LIN {X -0.018,Y -257.062,Z 1664.281,A 0.000,B 0.000,C 90.000,E1 50.598} C_DIS
LIN {X 0.149,Y -245.227,Z 1664.263,A 0.000,B 0.000,C 90.000,E1 47.310} C_DIS
LIN {X -0.032,Y -234.510,Z 1664.245,A 0.000,B 0.000,C 90.000,E1 44.028} C_DIS
LIN {X 0.021,Y -224.506,Z 1664.226,A 0.000,B 0.000,C 90.000,E1 40.620} C_DIS
LIN {X -0.056,Y -216.375,Z 1664.209,A 0.000,B 0.000,C 90.000,E1 37.569} C_DIS
LIN {X 0.091,Y -208.880,Z 1664.191,A 0.000,B 0.000,C 90.000,E1 34.405} C_DIS
LIN {X -0.009,Y -201.954,Z 1664.174,A 0.000,B 0.000,C 90.000,E1 31.258} C_DIS
LIN {X 0.029,Y -195.573,Z 1664.156,A 0.000,B 0.000,C 90.000,E1 28.025} C_DIS
LIN {X -0.014,Y -189.790,Z 1664.138,A 0.000,B 0.000,C 90.000,E1 24.771} C_DIS
LIN {X -0.011,Y -184.718,Z 1664.119,A 0.000,B 0.000,C 90.000,E1 21.461} C_DIS
LIN {X -0.051,Y -180.294,Z 1664.101,A 0.000,B 0.000,C 90.000,E1 18.127} C_DIS
LIN {X 0.041,Y -176.550,Z 1664.082,A 0.000,B 0.000,C 90.000,E1 14.717} C_DIS
LIN {X -0.073,Y -172.830,Z 1664.058,A 0.000,B 0.000,C 90.000,E1 10.489} C_DIS
LIN {X 0.072,Y -169.604,Z 1664.029,A 0.000,B 0.000,C 90.000,E1 5.277} C_DIS
LIN {X -0.060,Y -167.411,Z 1663.993,A 0.000,B 0.000,C 90.000,E1 358.682} C_DIS
LIN {X -0.010,Y -168.408,Z 1663.930,A 0.000,B 0.000,C 90.000,E1 347.353} C_DIS
LIN {X 0.070,Y -171.194,Z 1663.901,A 0.000,B 0.000,C 90.000,E1 342.127} C_DIS
LIN {X -0.005,Y -174.815,Z 1663.877,A 0.000,B 0.000,C 90.000,E1 337.847} C_DIS
LIN {X 0.066,Y -178.691,Z 1663.858,A 0.000,B 0.000,C 90.000,E1 334.409} C_DIS
LIN {X -0.019,Y -183.314,Z 1663.839,A 0.000,B 0.000,C 90.000,E1 331.051} C_DIS
LIN {X -0.041,Y -188.766,Z 1663.821,A 0.000,B 0.000,C 90.000,E1 327.709} C_DIS
LIN {X 0.106,Y -193.563,Z 1663.807,A 0.000,B 0.000,C 90.000,E1 325.182} C_DIS
LIN {X -0.026,Y -198.905,Z 1663.793,A 0.000,B 0.000,C 90.000,E1 322.763} C_DIS
LIN {X 0.074,Y -205.972,Z 1663.777,A 0.000,B 0.000,C 90.000,E1 319.908} C_DIS
LIN {X 0.004,Y -213.943,Z 1663.762,A 0.000,B 0.000,C 90.000,E1 317.148} C_DIS
LIN {X -0.055,Y -222.887,Z 1663.747,A 0.000,B 0.000,C 90.000,E1 314.433} C_DIS
LIN {X 0.034,Y -234.369,Z 1663.730,A 0.000,B 0.000,C 90.000,E1 311.353} C_DIS
LIN {X -0.013,Y -245.664,Z 1663.715,A 0.000,B 0.000,C 90.000,E1 308.749} C_DIS
LIN {X -0.136,Y -256.628,Z 1663.703,A 0.000,B 0.000,C 90.000,E1 306.583} C_DIS
LIN {X -0.013,Y -272.944,Z 1663.687,A 0.000,B 0.000,C 90.000,E1 303.706} C_DIS
LIN {X 0.096,Y -291.059,Z 1663.672,A 0.000,B 0.000,C 90.000,E1 300.924} C_DIS
LIN {X -0.028,Y -310.502,Z 1663.657,A 0.000,B 0.000,C 90.000,E1 298.281} C_DIS
LIN {X -0.059,Y -323.099,Z 1663.648,A 0.000,B 0.000,C 90.000,E1 296.668} C_DIS
LIN {X -0.045,Y -335.406,Z 1663.639,A 0.000,B 0.000,C 90.000,E1 295.079} C_DIS
LIN {X 0.044,Y -350.168,Z 1663.629,A 0.000,B 0.000,C 90.000,E1 293.206} C_DIS
LIN {X -0.102,Y -362.395,Z 1663.621,A 0.000,B 0.000,C 90.000,E1 291.716} C_DIS
LIN {X 0.183,Y -371.921,Z 1663.614,A 0.000,B 0.000,C 90.000,E1 290.482} C_DIS
LIN {X -0.006,Y -378.695,Z 1663.609,A 0.000,B 0.000,C 90.000,E1 289.631} C_DIS
LIN {X -0.131,Y -384.956,Z 1663.604,A 0.000,B 0.000,C 90.000,E1 288.779} C_DIS
LIN {X 0.161,Y -390.546,Z 1663.599,A 0.000,B 0.000,C 90.000,E1 287.873} C_DIS
LIN {X 0.025,Y -395.292,Z 1663.595,A 0.000,B 0.000,C 90.000,E1 287.040} C_DIS
LIN {X -0.133,Y -398.011,Z 1663.592,A 0.000,B 0.000,C 90.000,E1 286.496} C_DIS
LIN {X 0.180,Y -401.321,Z 1663.587,A 0.000,B 0.000,C 90.000,E1 285.607} C_DIS
LIN {X 0.057,Y -403.082,Z 1663.584,A 0.000,B 0.000,C 90.000,E1 285.064} C_DIS
LIN {X -0.167,Y -404.505,Z 1663.581,A 0.000,B 0.000,C 90.000,E1 284.537} C_DIS
LIN {X 0.016,Y -405.481,Z 1663.578,A 0.000,B 0.000,C 90.000,E1 283.953} C_DIS
LIN {X -0.091,Y -406.070,Z 1663.574,A 0.000,B 0.000,C 90.000,E1 283.411} C_DIS
LIN {X 0.108,Y -406.200,Z 1663.571,A 0.000,B 0.000,C 90.000,E1 282.827} C_DIS
LIN {X -0.084,Y -405.886,Z 1663.568,A 0.000,B 0.000,C 90.000,E1 282.299} C_DIS
LIN {X 0.122,Y -405.095,Z 1663.565,A 0.000,B 0.000,C 90.000,E1 281.715} C_DIS
LIN {X -0.071,Y -403.731,Z 1663.562,A 0.000,B 0.000,C 90.000,E1 281.186} C_DIS
LIN {X 0.125,Y -401.822,Z 1663.559,A 0.000,B 0.000,C 90.000,E1 280.602} C_DIS
LIN {X -0.082,Y -399.374,Z 1663.556,A 0.000,B 0.000,C 90.000,E1 280.074} C_DIS
LIN {X 0.018,Y -396.298,Z 1663.553,A 0.000,B 0.000,C 90.000,E1 279.500} C_DIS
LIN {X -0.158,Y -390.804,Z 1663.548,A 0.000,B 0.000,C 90.000,E1 278.681} C_DIS
LIN {X -0.052,Y -384.534,Z 1663.543,A 0.000,B 0.000,C 90.000,E1 277.814} C_DIS
LIN {X -0.008,Y -377.358,Z 1663.539,A 0.000,B 0.000,C 90.000,E1 276.947} C_DIS
LIN {X 0.033,Y -371.956,Z 1663.535,A 0.000,B 0.000,C 90.000,E1 276.372} C_DIS
LIN {X -0.134,Y -366.148,Z 1663.532,A 0.000,B 0.000,C 90.000,E1 275.853} C_DIS
LIN {X -0.023,Y -359.968,Z 1663.530,A 0.000,B 0.000,C 90.000,E1 275.334} C_DIS
LIN {X 0.031,Y -353.523,Z 1663.527,A 0.000,B 0.000,C 90.000,E1 274.878} C_DIS
LIN {X 0.062,Y -347.074,Z 1663.525,A 0.000,B 0.000,C 90.000,E1 274.473} C_DIS
LIN {X -0.043,Y -337.427,Z 1663.522,A 0.000,B 0.000,C 90.000,E1 273.955} C_DIS
LIN {X 0.126,Y -327.816,Z 1663.519,A 0.000,B 0.000,C 90.000,E1 273.440} C_DIS
LIN {X -0.078,Y -318.091,Z 1663.517,A 0.000,B 0.000,C 90.000,E1 273.037} C_DIS
LIN {X -0.021,Y -308.209,Z 1663.515,A 0.000,B 0.000,C 90.000,E1 272.636} C_DIS
LIN {X -0.061,Y -301.352,Z 1663.513,A 0.000,B 0.000,C 90.000,E1 272.407} C_DIS
LIN {X 0.052,Y -294.071,Z 1663.512,A 0.000,B 0.000,C 90.000,E1 272.178} C_DIS
LIN {X 0.045,Y -286.541,Z 1663.511,A 0.000,B 0.000,C 90.000,E1 272.007} C_DIS
LIN {X -0.087,Y -277.923,Z 1663.510,A 0.000,B 0.000,C 90.000,E1 271.892} C_DIS
LIN {X -0.075,Y -267.107,Z 1663.510,A 0.000,B 0.000,C 90.000,E1 271.776} C_DIS
LIN {X -0.077,Y -233.599,Z 1663.509,A 0.000,B 0.000,C 90.000,E1 271.604} C_DIS
LIN {X -0.054,Y -181.975,Z 1663.508,A 0.000,B 0.000,C 90.000,E1 271.375} C_DIS
LIN {X -0.080,Y -181.381,Z 1663.507,A 0.000,B 0.000,C 90.000,E1 271.375} C_DIS
LIN {X -0.030,Y -181.572,Z 1663.502,A 0.000,B 0.000,C 90.000,E1 270.458} C_DIS
LIN {X -0.052,Y -180.906,Z 1663.474,A 0.000,B 0.000,C 90.000,E1 265.412} C_DIS
LIN {X 0.022,Y -180.702,Z 1663.470,A 0.000,B 0.000,C 90.000,E1 264.546} C_DIS
LIN {X -0.076,Y -178.788,Z 1663.442,A 0.000,B 0.000,C 90.000,E1 259.511} C_DIS
LIN {X 0.002,Y -175.834,Z 1663.413,A 0.000,B 0.000,C 90.000,E1 254.393} C_DIS
LIN {X 0.002,Y -172.023,Z 1663.385,A 0.000,B 0.000,C 90.000,E1 249.263} C_DIS
LIN {X -0.022,Y -171.447,Z 1663.380,A 0.000,B 0.000,C 90.000,E1 248.411} C_DIS
LIN {X 0.032,Y -167.682,Z 1663.356,A 0.000,B 0.000,C 90.000,E1 244.076} C_DIS
LIN {X -0.028,Y -166.359,Z 1663.346,A 0.000,B 0.000,C 90.000,E1 242.359} C_DIS
LIN {X -0.035,Y -163.092,Z 1663.327,A 0.000,B 0.000,C 90.000,E1 238.869} C_DIS
LIN {X 0.015,Y -161.036,Z 1663.312,A 0.000,B 0.000,C 90.000,E1 236.215} C_DIS
LIN {X -0.001,Y -157.775,Z 1663.293,A 0.000,B 0.000,C 90.000,E1 232.683} C_DIS
LIN {X 0.063,Y -155.812,Z 1663.278,A 0.000,B 0.000,C 90.000,E1 229.989} C_DIS
LIN {X 0.009,Y -152.063,Z 1663.253,A 0.000,B 0.000,C 90.000,E1 225.526} C_DIS
LIN {X -0.080,Y -150.314,Z 1663.238,A 0.000,B 0.000,C 90.000,E1 222.852} C_DIS
LIN {X 0.058,Y -147.058,Z 1663.213,A 0.000,B 0.000,C 90.000,E1 218.257} C_DIS
LIN {X 0.050,Y -145.634,Z 1663.197,A 0.000,B 0.000,C 90.000,E1 215.518} C_DIS
LIN {X 0.048,Y -143.017,Z 1663.172,A 0.000,B 0.000,C 90.000,E1 210.924} C_DIS
LIN {X -0.022,Y -141.644,Z 1663.151,A 0.000,B 0.000,C 90.000,E1 207.257} C_DIS
LIN {X 0.030,Y -139.440,Z 1663.115,A 0.000,B 0.000,C 90.000,E1 200.737} C_DIS
LIN {X -0.048,Y -139.174,Z 1663.105,A 0.000,B 0.000,C 90.000,E1 198.906} C_DIS
LIN {X -0.020,Y -138.318,Z 1663.053,A 0.000,B 0.000,C 90.000,E1 189.557} C_DIS
LIN {X -0.011,Y -139.471,Z 1663.006,A 0.000,B 0.000,C 90.000,E1 181.146} C_DIS
LIN {X 0.070,Y -141.043,Z 1662.975,A 0.000,B 0.000,C 90.000,E1 175.527} C_DIS
LIN {X 0.024,Y -142.413,Z 1662.960,A 0.000,B 0.000,C 90.000,E1 172.761} C_DIS
LIN {X -0.055,Y -144.647,Z 1662.934,A 0.000,B 0.000,C 90.000,E1 168.173} C_DIS
LIN {X 0.005,Y -147.843,Z 1662.909,A 0.000,B 0.000,C 90.000,E1 163.559} C_DIS
LIN {X -0.052,Y -150.541,Z 1662.888,A 0.000,B 0.000,C 90.000,E1 159.934} C_DIS
LIN {X -0.034,Y -154.007,Z 1662.868,A 0.000,B 0.000,C 90.000,E1 156.305} C_DIS
LIN {X 0.026,Y -157.421,Z 1662.848,A 0.000,B 0.000,C 90.000,E1 152.692} C_DIS
LIN {X 0.049,Y -161.632,Z 1662.829,A 0.000,B 0.000,C 90.000,E1 149.125} C_DIS
LIN {X 0.067,Y -165.828,Z 1662.809,A 0.000,B 0.000,C 90.000,E1 145.595} C_DIS
LIN {X 0.060,Y -170.798,Z 1662.790,A 0.000,B 0.000,C 90.000,E1 142.110} C_DIS
LIN {X -0.023,Y -175.669,Z 1662.771,A 0.000,B 0.000,C 90.000,E1 138.690} C_DIS
LIN {X 0.101,Y -181.282,Z 1662.752,A 0.000,B 0.000,C 90.000,E1 135.243} C_DIS
LIN {X -0.027,Y -186.760,Z 1662.733,A 0.000,B 0.000,C 90.000,E1 131.919} C_DIS
LIN {X 0.045,Y -191.355,Z 1662.719,A 0.000,B 0.000,C 90.000,E1 129.402} C_DIS
LIN {X -0.031,Y -197.192,Z 1662.701,A 0.000,B 0.000,C 90.000,E1 126.137} C_DIS
LIN {X 0.053,Y -200.469,Z 1662.692,A 0.000,B 0.000,C 90.000,E1 124.485} C_DIS
LIN {X 0.025,Y -207.457,Z 1662.671,A 0.000,B 0.000,C 90.000,E1 120.718} C_DIS
LIN {X 0.001,Y -328.831,Z 1662.671,A 0.000,B 0.000,C 90.000,E1 120.718} C_DIS
LIN {X 0.095,Y -335.276,Z 1662.669,A 0.000,B 0.000,C 90.000,E1 120.463} C_DIS
LIN {X 0.140,Y -338.242,Z 1662.668,A 0.000,B 0.000,C 90.000,E1 120.207} C_DIS
LIN {X 0.031,Y -341.943,Z 1662.665,A 0.000,B 0.000,C 90.000,E1 119.745} C_DIS
LIN {X -0.120,Y -343.606,Z 1662.664,A 0.000,B 0.000,C 90.000,E1 119.461} C_DIS
LIN {X -0.117,Y -357.433,Z 1662.647,A 0.000,B 0.000,C 90.000,E1 116.411} C_DIS
LIN {X 0.102,Y -371.411,Z 1662.632,A 0.000,B 0.000,C 90.000,E1 113.695} C_DIS
LIN {X -0.197,Y -385.182,Z 1662.619,A 0.000,B 0.000,C 90.000,E1 111.408} C_DIS
LIN {X 0.071,Y -400.321,Z 1662.606,A 0.000,B 0.000,C 90.000,E1 109.087} C_DIS
LIN {X 0.085,Y -416.932,Z 1662.594,A 0.000,B 0.000,C 90.000,E1 106.858} C_DIS
LIN {X -0.140,Y -435.129,Z 1662.582,A 0.000,B 0.000,C 90.000,E1 104.717} C_DIS
LIN {X 0.160,Y -454.786,Z 1662.570,A 0.000,B 0.000,C 90.000,E1 102.591} C_DIS
LIN {X 0.237,Y -475.081,Z 1662.559,A 0.000,B 0.000,C 90.000,E1 100.658} C_DIS
LIN {X -0.126,Y -501.079,Z 1662.547,A 0.000,B 0.000,C 90.000,E1 98.511} C_DIS
LIN {X 0.196,Y -504.675,Z 1662.545,A 0.000,B 0.000,C 90.000,E1 98.049} C_DIS
LIN {X 0.127,Y -506.032,Z 1662.543,A 0.000,B 0.000,C 90.000,E1 97.814} C_DIS
LIN {X -0.012,Y -507.029,Z 1662.542,A 0.000,B 0.000,C 90.000,E1 97.587} C_DIS
LIN {X -0.192,Y -508.132,Z 1662.539,A 0.000,B 0.000,C 90.000,E1 97.125} C_DIS
LIN {X 0.139,Y -508.201,Z 1662.537,A 0.000,B 0.000,C 90.000,E1 96.606} C_DIS
LIN {X -0.030,Y -507.247,Z 1662.534,A 0.000,B 0.000,C 90.000,E1 96.144} C_DIS
LIN {X -0.197,Y -505.098,Z 1662.531,A 0.000,B 0.000,C 90.000,E1 95.682} C_DIS
LIN {X 0.175,Y -494.734,Z 1662.523,A 0.000,B 0.000,C 90.000,E1 94.188} C_DIS
LIN {X -0.129,Y -484.275,Z 1662.515,A 0.000,B 0.000,C 90.000,E1 92.751} C_DIS
LIN {X -0.148,Y -473.595,Z 1662.507,A 0.000,B 0.000,C 90.000,E1 91.260} C_DIS
LIN {X 0.152,Y -459.135,Z 1662.496,A 0.000,B 0.000,C 90.000,E1 89.198} C_DIS
LIN {X 0.163,Y -448.105,Z 1662.487,A 0.000,B 0.000,C 90.000,E1 87.650} C_DIS
LIN {X -0.016,Y -436.597,Z 1662.478,A 0.000,B 0.000,C 90.000,E1 86.102} C_DIS
LIN {X -0.200,Y -423.089,Z 1662.468,A 0.000,B 0.000,C 90.000,E1 84.261} C_DIS
LIN {X 0.101,Y -404.171,Z 1662.453,A 0.000,B 0.000,C 90.000,E1 81.489} C_DIS
LIN {X -0.040,Y -386.478,Z 1662.437,A 0.000,B 0.000,C 90.000,E1 78.701} C_DIS
LIN {X -0.091,Y -371.265,Z 1662.423,A 0.000,B 0.000,C 90.000,E1 76.117} C_DIS
LIN {X -0.016,Y -356.575,Z 1662.408,A 0.000,B 0.000,C 90.000,E1 73.449} C_DIS
LIN {X -0.003,Y -339.651,Z 1662.390,A 0.000,B 0.000,C 90.000,E1 70.115} C_DIS
LIN {X 0.105,Y -328.061,Z 1662.376,A 0.000,B 0.000,C 90.000,E1 67.614} C_DIS
LIN {X -0.069,Y -315.627,Z 1662.360,A 0.000,B 0.000,C 90.000,E1 64.793} C_DIS
LIN {X -0.198,Y -304.785,Z 1662.345,A 0.000,B 0.000,C 90.000,E1 62.231} C_DIS
LIN {X 0.078,Y -296.635,Z 1662.335,A 0.000,B 0.000,C 90.000,E1 60.205} C_DIS
LIN {X 0.085,Y -288.273,Z 1662.323,A 0.000,B 0.000,C 90.000,E1 58.201} C_DIS
LIN {X 0.086,Y -279.642,Z 1662.312,A 0.000,B 0.000,C 90.000,E1 56.167} C_DIS
LIN {X 0.022,Y -268.032,Z 1662.297,A 0.000,B 0.000,C 90.000,E1 53.417} C_DIS
LIN {X 0.041,Y -255.522,Z 1662.279,A 0.000,B 0.000,C 90.000,E1 50.231} C_DIS
LIN {X -0.023,Y -243.854,Z 1662.261,A 0.000,B 0.000,C 90.000,E1 46.986} C_DIS
LIN {X 0.101,Y -233.249,Z 1662.242,A 0.000,B 0.000,C 90.000,E1 43.623} C_DIS
LIN {X 0.015,Y -224.374,Z 1662.226,A 0.000,B 0.000,C 90.000,E1 40.620} C_DIS
LIN {X 0.108,Y -216.225,Z 1662.209,A 0.000,B 0.000,C 90.000,E1 37.523} C_DIS
LIN {X 0.079,Y -208.720,Z 1662.191,A 0.000,B 0.000,C 90.000,E1 34.405} C_DIS
LIN {X -0.025,Y -201.781,Z 1662.174,A 0.000,B 0.000,C 90.000,E1 31.258} C_DIS
LIN {X 0.011,Y -195.398,Z 1662.156,A 0.000,B 0.000,C 90.000,E1 28.025} C_DIS
LIN {X -0.037,Y -189.641,Z 1662.138,A 0.000,B 0.000,C 90.000,E1 24.771} C_DIS
LIN {X -0.036,Y -184.606,Z 1662.119,A 0.000,B 0.000,C 90.000,E1 21.461} C_DIS
LIN {X -0.021,Y -180.218,Z 1662.101,A 0.000,B 0.000,C 90.000,E1 18.109} C_DIS
LIN {X -0.036,Y -175.705,Z 1662.077,A 0.000,B 0.000,C 90.000,E1 13.883} C_DIS
LIN {X -0.043,Y -172.203,Z 1662.053,A 0.000,B 0.000,C 90.000,E1 9.613} C_DIS
LIN {X 0.034,Y -169.193,Z 1662.025,A 0.000,B 0.000,C 90.000,E1 4.416} C_DIS
LIN {X 0.021,Y -167.142,Z 1661.978,A 0.000,B 0.000,C 90.000,E1 356.045} C_DIS
LIN {X 0.053,Y -168.789,Z 1661.925,A 0.000,B 0.000,C 90.000,E1 346.464} C_DIS
LIN {X 0.074,Y -171.244,Z 1661.901,A 0.000,B 0.000,C 90.000,E1 342.127} C_DIS
LIN {X 0.000,Y -174.891,Z 1661.877,A 0.000,B 0.000,C 90.000,E1 337.847} C_DIS
LIN {X 0.073,Y -178.787,Z 1661.858,A 0.000,B 0.000,C 90.000,E1 334.409} C_DIS
LIN {X -0.009,Y -183.433,Z 1661.839,A 0.000,B 0.000,C 90.000,E1 331.051} C_DIS
LIN {X -0.027,Y -188.918,Z 1661.821,A 0.000,B 0.000,C 90.000,E1 327.709} C_DIS
LIN {X -0.036,Y -193.733,Z 1661.807,A 0.000,B 0.000,C 90.000,E1 325.229} C_DIS
LIN {X -0.006,Y -199.082,Z 1661.793,A 0.000,B 0.000,C 90.000,E1 322.763} C_DIS
LIN {X 0.100,Y -206.138,Z 1661.777,A 0.000,B 0.000,C 90.000,E1 319.908} C_DIS
LIN {X 0.033,Y -214.113,Z 1661.762,A 0.000,B 0.000,C 90.000,E1 317.148} C_DIS
LIN {X -0.021,Y -223.045,Z 1661.747,A 0.000,B 0.000,C 90.000,E1 314.433} C_DIS
LIN {X -0.080,Y -234.501,Z 1661.730,A 0.000,B 0.000,C 90.000,E1 311.391} C_DIS
LIN {X 0.032,Y -245.793,Z 1661.715,A 0.000,B 0.000,C 90.000,E1 308.749} C_DIS
LIN {X -0.103,Y -254.812,Z 1661.705,A 0.000,B 0.000,C 90.000,E1 306.950} C_DIS
LIN {X 0.064,Y -268.784,Z 1661.691,A 0.000,B 0.000,C 90.000,E1 304.405} C_DIS
LIN {X -0.125,Y -284.119,Z 1661.678,A 0.000,B 0.000,C 90.000,E1 302.005} C_DIS
LIN {X -0.034,Y -300.650,Z 1661.665,A 0.000,B 0.000,C 90.000,E1 299.617} C_DIS
LIN {X 0.029,Y -318.190,Z 1661.652,A 0.000,B 0.000,C 90.000,E1 297.308} C_DIS
LIN {X -0.073,Y -333.022,Z 1661.641,A 0.000,B 0.000,C 90.000,E1 295.412} C_DIS
LIN {X 0.113,Y -347.706,Z 1661.631,A 0.000,B 0.000,C 90.000,E1 293.515} C_DIS
LIN {X -0.078,Y -359.926,Z 1661.622,A 0.000,B 0.000,C 90.000,E1 292.025} C_DIS
LIN {X -0.083,Y -371.883,Z 1661.614,A 0.000,B 0.000,C 90.000,E1 290.536} C_DIS
LIN {X 0.076,Y -378.655,Z 1661.609,A 0.000,B 0.000,C 90.000,E1 289.631} C_DIS
LIN {X -0.047,Y -384.908,Z 1661.604,A 0.000,B 0.000,C 90.000,E1 288.779} C_DIS
LIN {X -0.126,Y -390.518,Z 1661.599,A 0.000,B 0.000,C 90.000,E1 287.928} C_DIS
LIN {X 0.110,Y -395.292,Z 1661.595,A 0.000,B 0.000,C 90.000,E1 287.040} C_DIS
LIN {X -0.047,Y -398.020,Z 1661.592,A 0.000,B 0.000,C 90.000,E1 286.496} C_DIS
LIN {X -0.120,Y -401.353,Z 1661.587,A 0.000,B 0.000,C 90.000,E1 285.662} C_DIS
LIN {X 0.144,Y -403.152,Z 1661.584,A 0.000,B 0.000,C 90.000,E1 285.064} C_DIS
LIN {X -0.079,Y -404.572,Z 1661.581,A 0.000,B 0.000,C 90.000,E1 284.537} C_DIS
LIN {X 0.104,Y -405.619,Z 1661.578,A 0.000,B 0.000,C 90.000,E1 283.953} C_DIS
LIN {X -0.002,Y -406.199,Z 1661.574,A 0.000,B 0.000,C 90.000,E1 283.411} C_DIS
LIN {X 0.198,Y -406.365,Z 1661.571,A 0.000,B 0.000,C 90.000,E1 282.827} C_DIS
LIN {X 0.007,Y -406.061,Z 1661.568,A 0.000,B 0.000,C 90.000,E1 282.299} C_DIS
LIN {X -0.184,Y -405.249,Z 1661.565,A 0.000,B 0.000,C 90.000,E1 281.771} C_DIS
LIN {X 0.020,Y -403.898,Z 1661.562,A 0.000,B 0.000,C 90.000,E1 281.186} C_DIS
LIN {X -0.177,Y -402.005,Z 1661.559,A 0.000,B 0.000,C 90.000,E1 280.658} C_DIS
LIN {X 0.011,Y -399.538,Z 1661.556,A 0.000,B 0.000,C 90.000,E1 280.074} C_DIS
LIN {X 0.111,Y -396.458,Z 1661.553,A 0.000,B 0.000,C 90.000,E1 279.500} C_DIS
LIN {X -0.065,Y -390.923,Z 1661.548,A 0.000,B 0.000,C 90.000,E1 278.681} C_DIS
LIN {X 0.042,Y -384.616,Z 1661.543,A 0.000,B 0.000,C 90.000,E1 277.814} C_DIS
LIN {X 0.084,Y -377.417,Z 1661.539,A 0.000,B 0.000,C 90.000,E1 276.947} C_DIS
LIN {X 0.119,Y -371.993,Z 1661.536,A 0.000,B 0.000,C 90.000,E1 276.372} C_DIS
LIN {X -0.064,Y -366.160,Z 1661.532,A 0.000,B 0.000,C 90.000,E1 275.853} C_DIS
LIN {X 0.051,Y -359.946,Z 1661.530,A 0.000,B 0.000,C 90.000,E1 275.334} C_DIS
LIN {X 0.125,Y -353.500,Z 1661.527,A 0.000,B 0.000,C 90.000,E1 274.878} C_DIS
LIN {X 0.080,Y -343.781,Z 1661.524,A 0.000,B 0.000,C 90.000,E1 274.302} C_DIS
LIN {X -0.132,Y -334.628,Z 1661.521,A 0.000,B 0.000,C 90.000,E1 273.841} C_DIS
LIN {X 0.079,Y -324.911,Z 1661.519,A 0.000,B 0.000,C 90.000,E1 273.326} C_DIS
LIN {X -0.052,Y -315.071,Z 1661.516,A 0.000,B 0.000,C 90.000,E1 272.922} C_DIS
LIN {X 0.061,Y -304.968,Z 1661.514,A 0.000,B 0.000,C 90.000,E1 272.522} C_DIS
LIN {X 0.103,Y -297.928,Z 1661.513,A 0.000,B 0.000,C 90.000,E1 272.293} C_DIS
LIN {X -0.025,Y -290.295,Z 1661.512,A 0.000,B 0.000,C 90.000,E1 272.121} C_DIS
LIN {X 0.019,Y -281.682,Z 1661.511,A 0.000,B 0.000,C 90.000,E1 271.949} C_DIS
LIN {X -0.034,Y -272.063,Z 1661.510,A 0.000,B 0.000,C 90.000,E1 271.835} C_DIS
LIN {X -0.069,Y -243.458,Z 1661.509,A 0.000,B 0.000,C 90.000,E1 271.661} C_DIS
LIN {X 0.071,Y -190.113,Z 1661.508,A 0.000,B 0.000,C 90.000,E1 271.375} C_DIS
LIN {X 0.009,Y -183.846,Z 1661.508,A 0.000,B 0.000,C 90.000,E1 271.375} C_DIS
LIN {X -0.011,Y -181.377,Z 1661.508,A 0.000,B 0.000,C 90.000,E1 271.375} C_DIS
LIN {X 0.042,Y -181.579,Z 1661.502,A 0.000,B 0.000,C 90.000,E1 270.344} C_DIS
LIN {X 0.046,Y -180.887,Z 1661.473,A 0.000,B 0.000,C 90.000,E1 265.122} C_DIS
LIN {X -0.070,Y -179.009,Z 1661.445,A 0.000,B 0.000,C 90.000,E1 260.095} C_DIS
LIN {X 0.024,Y -178.625,Z 1661.440,A 0.000,B 0.000,C 90.000,E1 259.218} C_DIS
LIN {X -0.078,Y -175.677,Z 1661.412,A 0.000,B 0.000,C 90.000,E1 254.157} C_DIS
LIN {X -0.065,Y -172.393,Z 1661.388,A 0.000,B 0.000,C 90.000,E1 249.880} C_DIS
LIN {X -0.049,Y -171.199,Z 1661.379,A 0.000,B 0.000,C 90.000,E1 248.156} C_DIS
LIN {X 0.002,Y -167.487,Z 1661.355,A 0.000,B 0.000,C 90.000,E1 243.819} C_DIS
LIN {X 0.010,Y -166.883,Z 1661.350,A 0.000,B 0.000,C 90.000,E1 242.948} C_DIS
LIN {X 0.001,Y -162.190,Z 1661.321,A 0.000,B 0.000,C 90.000,E1 237.709} C_DIS
LIN {X -0.032,Y -160.758,Z 1661.311,A 0.000,B 0.000,C 90.000,E1 235.960} C_DIS
LIN {X 0.036,Y -157.556,Z 1661.291,A 0.000,B 0.000,C 90.000,E1 232.396} C_DIS
LIN {X -0.025,Y -155.585,Z 1661.276,A 0.000,B 0.000,C 90.000,E1 229.747} C_DIS
LIN {X 0.027,Y -151.869,Z 1661.251,A 0.000,B 0.000,C 90.000,E1 225.243} C_DIS
LIN {X 0.040,Y -150.093,Z 1661.236,A 0.000,B 0.000,C 90.000,E1 222.528} C_DIS
LIN {X -0.043,Y -146.893,Z 1661.211,A 0.000,B 0.000,C 90.000,E1 218.016} C_DIS
LIN {X 0.062,Y -145.480,Z 1661.196,A 0.000,B 0.000,C 90.000,E1 215.231} C_DIS
LIN {X -0.022,Y -142.890,Z 1661.170,A 0.000,B 0.000,C 90.000,E1 210.669} C_DIS
LIN {X 0.035,Y -141.509,Z 1661.150,A 0.000,B 0.000,C 90.000,E1 206.950} C_DIS
LIN {X -0.047,Y -139.391,Z 1661.114,A 0.000,B 0.000,C 90.000,E1 200.482} C_DIS
LIN {X 0.004,Y -139.099,Z 1661.103,A 0.000,B 0.000,C 90.000,E1 198.598} C_DIS
LIN {X -0.005,Y -138.354,Z 1661.057,A 0.000,B 0.000,C 90.000,E1 190.197} C_DIS
LIN {X -0.011,Y -139.515,Z 1661.005,A 0.000,B 0.000,C 90.000,E1 180.859} C_DIS
LIN {X -0.071,Y -141.165,Z 1660.974,A 0.000,B 0.000,C 90.000,E1 175.298} C_DIS
LIN {X 0.041,Y -142.545,Z 1660.958,A 0.000,B 0.000,C 90.000,E1 172.470} C_DIS
LIN {X -0.034,Y -144.818,Z 1660.933,A 0.000,B 0.000,C 90.000,E1 167.881} C_DIS
LIN {X -0.047,Y -147.440,Z 1660.912,A 0.000,B 0.000,C 90.000,E1 164.212} C_DIS
LIN {X -0.018,Y -150.020,Z 1660.892,A 0.000,B 0.000,C 90.000,E1 160.550} C_DIS
LIN {X -0.012,Y -153.355,Z 1660.872,A 0.000,B 0.000,C 90.000,E1 156.922} C_DIS
LIN {X 0.037,Y -155.888,Z 1660.857,A 0.000,B 0.000,C 90.000,E1 154.204} C_DIS
LIN {X -0.064,Y -159.747,Z 1660.837,A 0.000,B 0.000,C 90.000,E1 150.667} C_DIS
LIN {X 0.002,Y -161.986,Z 1660.827,A 0.000,B 0.000,C 90.000,E1 148.869} C_DIS
LIN {X 0.021,Y -166.178,Z 1660.807,A 0.000,B 0.000,C 90.000,E1 145.341} C_DIS
LIN {X 0.014,Y -171.193,Z 1660.788,A 0.000,B 0.000,C 90.000,E1 141.859} C_DIS
LIN {X 0.044,Y -176.075,Z 1660.769,A 0.000,B 0.000,C 90.000,E1 138.405} C_DIS
LIN {X -0.093,Y -180.334,Z 1660.755,A 0.000,B 0.000,C 90.000,E1 135.891} C_DIS
LIN {X 0.015,Y -185.744,Z 1660.736,A 0.000,B 0.000,C 90.000,E1 132.486} C_DIS
LIN {X -0.071,Y -190.355,Z 1660.722,A 0.000,B 0.000,C 90.000,E1 130.011} C_DIS
LIN {X -0.025,Y -197.680,Z 1660.699,A 0.000,B 0.000,C 90.000,E1 125.884} C_DIS
LIN {X 0.017,Y -200.932,Z 1660.690,A 0.000,B 0.000,C 90.000,E1 124.246} C_DIS
LIN {X -0.009,Y -207.317,Z 1660.671,A 0.000,B 0.000,C 90.000,E1 120.797} C_DIS
LIN {X 0.051,Y -207.383,Z 1660.671,A 0.000,B 0.000,C 90.000,E1 120.747} C_DIS
LIN {X 0.036,Y -328.953,Z 1660.671,A 0.000,B 0.000,C 90.000,E1 120.747} C_DIS
LIN {X 0.114,Y -329.958,Z 1660.671,A 0.000,B 0.000,C 90.000,E1 120.718} C_DIS
LIN {X 0.136,Y -335.536,Z 1660.669,A 0.000,B 0.000,C 90.000,E1 120.463} C_DIS
LIN {X -0.134,Y -338.393,Z 1660.668,A 0.000,B 0.000,C 90.000,E1 120.256} C_DIS
LIN {X -0.073,Y -342.089,Z 1660.665,A 0.000,B 0.000,C 90.000,E1 119.745} C_DIS
LIN {X 0.074,Y -343.680,Z 1660.663,A 0.000,B 0.000,C 90.000,E1 119.411} C_DIS
LIN {X 0.057,Y -356.036,Z 1660.648,A 0.000,B 0.000,C 90.000,E1 116.668} C_DIS
LIN {X -0.090,Y -369.848,Z 1660.633,A 0.000,B 0.000,C 90.000,E1 114.003} C_DIS
LIN {X -0.080,Y -383.463,Z 1660.620,A 0.000,B 0.000,C 90.000,E1 111.663} C_DIS
LIN {X -0.221,Y -398.435,Z 1660.608,A 0.000,B 0.000,C 90.000,E1 109.396} C_DIS
LIN {X -0.138,Y -414.866,Z 1660.595,A 0.000,B 0.000,C 90.000,E1 107.149} C_DIS
LIN {X -0.012,Y -432.869,Z 1660.583,A 0.000,B 0.000,C 90.000,E1 104.954} C_DIS
LIN {X 0.180,Y -452.393,Z 1660.571,A 0.000,B 0.000,C 90.000,E1 102.827} C_DIS
LIN {X 0.099,Y -472.623,Z 1660.561,A 0.000,B 0.000,C 90.000,E1 100.894} C_DIS
LIN {X -0.103,Y -496.009,Z 1660.549,A 0.000,B 0.000,C 90.000,E1 98.916} C_DIS
LIN {X -0.235,Y -501.157,Z 1660.547,A 0.000,B 0.000,C 90.000,E1 98.511} C_DIS
LIN {X 0.042,Y -504.671,Z 1660.545,A 0.000,B 0.000,C 90.000,E1 98.049} C_DIS
LIN {X -0.027,Y -505.980,Z 1660.543,A 0.000,B 0.000,C 90.000,E1 97.814} C_DIS
LIN {X -0.166,Y -506.937,Z 1660.542,A 0.000,B 0.000,C 90.000,E1 97.587} C_DIS
LIN {X 0.158,Y -507.974,Z 1660.539,A 0.000,B 0.000,C 90.000,E1 97.068} C_DIS
LIN {X -0.016,Y -507.982,Z 1660.537,A 0.000,B 0.000,C 90.000,E1 96.606} C_DIS
LIN {X -0.185,Y -506.962,Z 1660.534,A 0.000,B 0.000,C 90.000,E1 96.144} C_DIS
LIN {X 0.260,Y -506.020,Z 1660.533,A 0.000,B 0.000,C 90.000,E1 95.853} C_DIS
LIN {X 0.149,Y -504.729,Z 1660.531,A 0.000,B 0.000,C 90.000,E1 95.625} C_DIS
LIN {X -0.090,Y -492.600,Z 1660.522,A 0.000,B 0.000,C 90.000,E1 93.955} C_DIS
LIN {X 0.029,Y -482.137,Z 1660.514,A 0.000,B 0.000,C 90.000,E1 92.465} C_DIS
LIN {X -0.029,Y -471.413,Z 1660.505,A 0.000,B 0.000,C 90.000,E1 90.974} C_DIS
LIN {X -0.021,Y -458.773,Z 1660.495,A 0.000,B 0.000,C 90.000,E1 89.198} C_DIS
LIN {X -0.012,Y -447.719,Z 1660.487,A 0.000,B 0.000,C 90.000,E1 87.650} C_DIS
LIN {X -0.193,Y -436.172,Z 1660.478,A 0.000,B 0.000,C 90.000,E1 86.102} C_DIS
LIN {X -0.076,Y -424.584,Z 1660.469,A 0.000,B 0.000,C 90.000,E1 84.489} C_DIS
LIN {X -0.189,Y -405.561,Z 1660.454,A 0.000,B 0.000,C 90.000,E1 81.781} C_DIS
LIN {X 0.175,Y -387.752,Z 1660.439,A 0.000,B 0.000,C 90.000,E1 78.926} C_DIS
LIN {X 0.065,Y -374.151,Z 1660.426,A 0.000,B 0.000,C 90.000,E1 76.645} C_DIS
LIN {X -0.189,Y -360.966,Z 1660.413,A 0.000,B 0.000,C 90.000,E1 74.338} C_DIS
LIN {X 0.172,Y -345.237,Z 1660.396,A 0.000,B 0.000,C 90.000,E1 71.275} C_DIS
LIN {X -0.034,Y -331.952,Z 1660.381,A 0.000,B 0.000,C 90.000,E1 68.539} C_DIS
LIN {X 0.137,Y -317.926,Z 1660.363,A 0.000,B 0.000,C 90.000,E1 65.357} C_DIS
LIN {X 0.017,Y -308.426,Z 1660.351,A 0.000,B 0.000,C 90.000,E1 63.127} C_DIS
LIN {X -0.024,Y -298.982,Z 1660.338,A 0.000,B 0.000,C 90.000,E1 60.845} C_DIS
LIN {X -0.115,Y -290.680,Z 1660.327,A 0.000,B 0.000,C 90.000,E1 58.869} C_DIS
LIN {X -0.060,Y -282.122,Z 1660.316,A 0.000,B 0.000,C 90.000,E1 56.834} C_DIS
LIN {X 0.081,Y -271.922,Z 1660.302,A 0.000,B 0.000,C 90.000,E1 54.402} C_DIS
LIN {X -0.007,Y -260.592,Z 1660.287,A 0.000,B 0.000,C 90.000,E1 51.618} C_DIS
LIN {X -0.070,Y -248.599,Z 1660.269,A 0.000,B 0.000,C 90.000,E1 48.405} C_DIS
LIN {X 0.020,Y -237.594,Z 1660.250,A 0.000,B 0.000,C 90.000,E1 45.081} C_DIS
LIN {X 0.031,Y -228.427,Z 1660.234,A 0.000,B 0.000,C 90.000,E1 42.081} C_DIS
LIN {X 0.013,Y -219.921,Z 1660.217,A 0.000,B 0.000,C 90.000,E1 39.036} C_DIS
LIN {X 0.028,Y -212.085,Z 1660.200,A 0.000,B 0.000,C 90.000,E1 35.931} C_DIS
LIN {X 0.119,Y -204.857,Z 1660.182,A 0.000,B 0.000,C 90.000,E1 32.752} C_DIS
LIN {X -0.016,Y -198.220,Z 1660.164,A 0.000,B 0.000,C 90.000,E1 29.589} C_DIS
LIN {X -0.081,Y -192.191,Z 1660.146,A 0.000,B 0.000,C 90.000,E1 26.360} C_DIS
LIN {X 0.061,Y -186.832,Z 1660.128,A 0.000,B 0.000,C 90.000,E1 23.025} C_DIS
LIN {X 0.029,Y -182.155,Z 1660.109,A 0.000,B 0.000,C 90.000,E1 19.704} C_DIS
LIN {X 0.099,Y -178.184,Z 1660.091,A 0.000,B 0.000,C 90.000,E1 16.315} C_DIS
LIN {X -0.065,Y -174.163,Z 1660.067,A 0.000,B 0.000,C 90.000,E1 12.119} C_DIS
LIN {X -0.013,Y -171.065,Z 1660.043,A 0.000,B 0.000,C 90.000,E1 7.814} C_DIS
LIN {X -0.031,Y -168.499,Z 1660.015,A 0.000,B 0.000,C 90.000,E1 2.636} C_DIS
LIN {X -0.017,Y -167.124,Z 1659.968,A 0.000,B 0.000,C 90.000,E1 354.318} C_DIS
LIN {X 0.056,Y -168.825,Z 1659.925,A 0.000,B 0.000,C 90.000,E1 346.464} C_DIS
LIN {X 0.043,Y -171.926,Z 1659.896,A 0.000,B 0.000,C 90.000,E1 341.275} C_DIS
LIN {X 0.057,Y -175.869,Z 1659.872,A 0.000,B 0.000,C 90.000,E1 336.975} C_DIS
LIN {X -0.009,Y -179.979,Z 1659.853,A 0.000,B 0.000,C 90.000,E1 333.589} C_DIS
LIN {X 0.019,Y -184.867,Z 1659.834,A 0.000,B 0.000,C 90.000,E1 330.205} C_DIS
LIN {X -0.024,Y -190.585,Z 1659.816,A 0.000,B 0.000,C 90.000,E1 326.882} C_DIS
LIN {X 0.021,Y -197.407,Z 1659.798,A 0.000,B 0.000,C 90.000,E1 323.577} C_DIS
LIN {X 0.080,Y -204.208,Z 1659.782,A 0.000,B 0.000,C 90.000,E1 320.723} C_DIS
LIN {X -0.013,Y -211.919,Z 1659.766,A 0.000,B 0.000,C 90.000,E1 317.957} C_DIS
LIN {X -0.123,Y -220.528,Z 1659.751,A 0.000,B 0.000,C 90.000,E1 315.243} C_DIS
LIN {X 0.061,Y -231.680,Z 1659.734,A 0.000,B 0.000,C 90.000,E1 312.123} C_DIS
LIN {X -0.022,Y -240.921,Z 1659.722,A 0.000,B 0.000,C 90.000,E1 309.886} C_DIS
LIN {X 0.077,Y -251.190,Z 1659.709,A 0.000,B 0.000,C 90.000,E1 307.649} C_DIS
LIN {X -0.053,Y -264.715,Z 1659.695,A 0.000,B 0.000,C 90.000,E1 305.152} C_DIS
LIN {X -0.019,Y -281.884,Z 1659.680,A 0.000,B 0.000,C 90.000,E1 302.339} C_DIS
LIN {X 0.033,Y -298.288,Z 1659.666,A 0.000,B 0.000,C 90.000,E1 299.951} C_DIS
LIN {X -0.048,Y -318.256,Z 1659.652,A 0.000,B 0.000,C 90.000,E1 297.334} C_DIS
LIN {X 0.040,Y -330.588,Z 1659.643,A 0.000,B 0.000,C 90.000,E1 295.720} C_DIS
LIN {X 0.048,Y -342.808,Z 1659.634,A 0.000,B 0.000,C 90.000,E1 294.155} C_DIS
LIN {X -0.077,Y -355.066,Z 1659.626,A 0.000,B 0.000,C 90.000,E1 292.642} C_DIS
LIN {X 0.186,Y -367.110,Z 1659.617,A 0.000,B 0.000,C 90.000,E1 291.099} C_DIS
LIN {X -0.045,Y -374.152,Z 1659.612,A 0.000,B 0.000,C 90.000,E1 290.248} C_DIS
LIN {X -0.209,Y -380.732,Z 1659.608,A 0.000,B 0.000,C 90.000,E1 289.396} C_DIS
LIN {X 0.043,Y -386.803,Z 1659.603,A 0.000,B 0.000,C 90.000,E1 288.489} C_DIS
LIN {X -0.007,Y -392.170,Z 1659.598,A 0.000,B 0.000,C 90.000,E1 287.638} C_DIS
LIN {X -0.134,Y -396.718,Z 1659.593,A 0.000,B 0.000,C 90.000,E1 286.804} C_DIS
LIN {X 0.100,Y -399.271,Z 1659.590,A 0.000,B 0.000,C 90.000,E1 286.205} C_DIS
LIN {X -0.033,Y -401.445,Z 1659.587,A 0.000,B 0.000,C 90.000,E1 285.662} C_DIS
LIN {X 0.127,Y -403.230,Z 1659.584,A 0.000,B 0.000,C 90.000,E1 285.079} C_DIS
LIN {X 0.010,Y -404.661,Z 1659.581,A 0.000,B 0.000,C 90.000,E1 284.537} C_DIS
LIN {X -0.201,Y -405.731,Z 1659.578,A 0.000,B 0.000,C 90.000,E1 284.008} C_DIS
LIN {X 0.088,Y -406.321,Z 1659.575,A 0.000,B 0.000,C 90.000,E1 283.411} C_DIS
LIN {X -0.107,Y -406.514,Z 1659.572,A 0.000,B 0.000,C 90.000,E1 282.883} C_DIS
LIN {X 0.098,Y -406.216,Z 1659.568,A 0.000,B 0.000,C 90.000,E1 282.299} C_DIS
LIN {X -0.092,Y -405.417,Z 1659.565,A 0.000,B 0.000,C 90.000,E1 281.771} C_DIS
LIN {X 0.113,Y -404.101,Z 1659.562,A 0.000,B 0.000,C 90.000,E1 281.186} C_DIS
LIN {X -0.084,Y -402.232,Z 1659.559,A 0.000,B 0.000,C 90.000,E1 280.658} C_DIS
LIN {X 0.105,Y -399.741,Z 1659.556,A 0.000,B 0.000,C 90.000,E1 280.074} C_DIS
LIN {X -0.186,Y -396.645,Z 1659.553,A 0.000,B 0.000,C 90.000,E1 279.557} C_DIS
LIN {X 0.030,Y -391.017,Z 1659.548,A 0.000,B 0.000,C 90.000,E1 278.681} C_DIS
LIN {X 0.136,Y -384.673,Z 1659.544,A 0.000,B 0.000,C 90.000,E1 277.814} C_DIS
LIN {X 0.177,Y -377.484,Z 1659.539,A 0.000,B 0.000,C 90.000,E1 276.947} C_DIS
LIN {X -0.132,Y -372.098,Z 1659.536,A 0.000,B 0.000,C 90.000,E1 276.429} C_DIS
LIN {X 0.122,Y -366.377,Z 1659.533,A 0.000,B 0.000,C 90.000,E1 275.853} C_DIS
LIN {X -0.083,Y -360.220,Z 1659.530,A 0.000,B 0.000,C 90.000,E1 275.391} C_DIS
LIN {X -0.008,Y -353.811,Z 1659.527,A 0.000,B 0.000,C 90.000,E1 274.935} C_DIS
LIN {X -0.063,Y -344.090,Z 1659.524,A 0.000,B 0.000,C 90.000,E1 274.359} C_DIS
LIN {X -0.046,Y -334.607,Z 1659.521,A 0.000,B 0.000,C 90.000,E1 273.841} C_DIS
LIN {X 0.154,Y -324.864,Z 1659.519,A 0.000,B 0.000,C 90.000,E1 273.326} C_DIS
LIN {X 0.004,Y -314.933,Z 1659.516,A 0.000,B 0.000,C 90.000,E1 272.922} C_DIS
LIN {X 0.106,Y -304.702,Z 1659.514,A 0.000,B 0.000,C 90.000,E1 272.522} C_DIS
LIN {X -0.140,Y -297.619,Z 1659.513,A 0.000,B 0.000,C 90.000,E1 272.350} C_DIS
LIN {X 0.052,Y -290.019,Z 1659.512,A 0.000,B 0.000,C 90.000,E1 272.121} C_DIS
LIN {X 0.112,Y -281.534,Z 1659.511,A 0.000,B 0.000,C 90.000,E1 271.949} C_DIS
LIN {X 0.055,Y -271.709,Z 1659.510,A 0.000,B 0.000,C 90.000,E1 271.835} C_DIS
LIN {X -0.071,Y -240.000,Z 1659.509,A 0.000,B 0.000,C 90.000,E1 271.661} C_DIS
LIN {X -0.059,Y -191.863,Z 1659.508,A 0.000,B 0.000,C 90.000,E1 271.432} C_DIS
LIN {X 0.046,Y -182.812,Z 1659.508,A 0.000,B 0.000,C 90.000,E1 271.375} C_DIS
LIN {X 0.026,Y -181.374,Z 1659.508,A 0.000,B 0.000,C 90.000,E1 271.375} C_DIS
LIN {X -0.057,Y -181.566,Z 1659.503,A 0.000,B 0.000,C 90.000,E1 270.516} C_DIS
LIN {X -0.067,Y -181.120,Z 1659.489,A 0.000,B 0.000,C 90.000,E1 267.993} C_DIS
LIN {X -0.078,Y -180.906,Z 1659.475,A 0.000,B 0.000,C 90.000,E1 265.469} C_DIS
LIN {X -0.022,Y -180.726,Z 1659.470,A 0.000,B 0.000,C 90.000,E1 264.609} C_DIS
LIN {X 0.076,Y -178.813,Z 1659.442,A 0.000,B 0.000,C 90.000,E1 259.511} C_DIS
LIN {X -0.018,Y -175.858,Z 1659.414,A 0.000,B 0.000,C 90.000,E1 254.448} C_DIS
LIN {X -0.035,Y -173.187,Z 1659.395,A 0.000,B 0.000,C 90.000,E1 251.040} C_DIS
LIN {X -0.034,Y -171.490,Z 1659.380,A 0.000,B 0.000,C 90.000,E1 248.465} C_DIS
LIN {X -0.046,Y -167.719,Z 1659.356,A 0.000,B 0.000,C 90.000,E1 244.152} C_DIS
LIN {X -0.030,Y -166.411,Z 1659.347,A 0.000,B 0.000,C 90.000,E1 242.410} C_DIS
LIN {X -0.031,Y -163.134,Z 1659.327,A 0.000,B 0.000,C 90.000,E1 238.918} C_DIS
LIN {X -0.065,Y -161.086,Z 1659.313,A 0.000,B 0.000,C 90.000,E1 236.294} C_DIS
LIN {X 0.044,Y -157.816,Z 1659.293,A 0.000,B 0.000,C 90.000,E1 232.718} C_DIS
LIN {X -0.018,Y -155.851,Z 1659.278,A 0.000,B 0.000,C 90.000,E1 230.070} C_DIS
LIN {X 0.038,Y -152.101,Z 1659.253,A 0.000,B 0.000,C 90.000,E1 225.567} C_DIS
LIN {X 0.057,Y -150.352,Z 1659.238,A 0.000,B 0.000,C 90.000,E1 222.852} C_DIS
LIN {X -0.014,Y -147.088,Z 1659.213,A 0.000,B 0.000,C 90.000,E1 218.338} C_DIS
LIN {X -0.020,Y -145.660,Z 1659.198,A 0.000,B 0.000,C 90.000,E1 215.598} C_DIS
LIN {X -0.016,Y -143.042,Z 1659.172,A 0.000,B 0.000,C 90.000,E1 211.003} C_DIS
LIN {X -0.015,Y -141.666,Z 1659.152,A 0.000,B 0.000,C 90.000,E1 207.308} C_DIS
LIN {X 0.029,Y -139.450,Z 1659.116,A 0.000,B 0.000,C 90.000,E1 200.791} C_DIS
LIN {X -0.050,Y -139.184,Z 1659.105,A 0.000,B 0.000,C 90.000,E1 198.960} C_DIS
LIN {X -0.027,Y -138.322,Z 1659.053,A 0.000,B 0.000,C 90.000,E1 189.613} C_DIS
LIN {X -0.020,Y -139.462,Z 1659.007,A 0.000,B 0.000,C 90.000,E1 181.203} C_DIS
LIN {X 0.061,Y -141.021,Z 1658.976,A 0.000,B 0.000,C 90.000,E1 175.584} C_DIS
LIN {X 0.016,Y -142.384,Z 1658.960,A 0.000,B 0.000,C 90.000,E1 172.818} C_DIS
LIN {X -0.063,Y -144.615,Z 1658.934,A 0.000,B 0.000,C 90.000,E1 168.229} C_DIS
LIN {X -0.002,Y -147.809,Z 1658.909,A 0.000,B 0.000,C 90.000,E1 163.614} C_DIS
LIN {X 0.086,Y -150.497,Z 1658.889,A 0.000,B 0.000,C 90.000,E1 159.934} C_DIS
LIN {X -0.035,Y -153.955,Z 1658.869,A 0.000,B 0.000,C 90.000,E1 156.357} C_DIS
LIN {X 0.028,Y -157.366,Z 1658.849,A 0.000,B 0.000,C 90.000,E1 152.743} C_DIS
LIN {X -0.030,Y -161.566,Z 1658.829,A 0.000,B 0.000,C 90.000,E1 149.203} C_DIS
LIN {X -0.017,Y -165.763,Z 1658.809,A 0.000,B 0.000,C 90.000,E1 145.674} C_DIS
LIN {X -0.032,Y -170.720,Z 1658.790,A 0.000,B 0.000,C 90.000,E1 142.190} C_DIS
LIN {X 0.012,Y -175.593,Z 1658.771,A 0.000,B 0.000,C 90.000,E1 138.728} C_DIS
LIN {X -0.001,Y -181.210,Z 1658.752,A 0.000,B 0.000,C 90.000,E1 135.324} C_DIS
LIN {X -0.009,Y -186.674,Z 1658.733,A 0.000,B 0.000,C 90.000,E1 131.962} C_DIS
LIN {X -0.065,Y -191.277,Z 1658.719,A 0.000,B 0.000,C 90.000,E1 129.483} C_DIS
LIN {X 0.014,Y -197.101,Z 1658.701,A 0.000,B 0.000,C 90.000,E1 126.171} C_DIS
LIN {X 0.051,Y -200.376,Z 1658.692,A 0.000,B 0.000,C 90.000,E1 124.532} C_DIS
LIN {X 0.039,Y -207.290,Z 1658.671,A 0.000,B 0.000,C 90.000,E1 120.797} C_DIS
LIN {X 0.020,Y -328.311,Z 1658.671,A 0.000,B 0.000,C 90.000,E1 120.797} C_DIS
LIN {X -0.067,Y -329.492,Z 1658.671,A 0.000,B 0.000,C 90.000,E1 120.797} C_DIS
LIN {X -0.095,Y -335.371,Z 1658.670,A 0.000,B 0.000,C 90.000,E1 120.541} C_DIS
LIN {X -0.035,Y -338.421,Z 1658.668,A 0.000,B 0.000,C 90.000,E1 120.256} C_DIS
LIN {X -0.019,Y -342.075,Z 1658.665,A 0.000,B 0.000,C 90.000,E1 119.745} C_DIS
LIN {X -0.024,Y -344.942,Z 1658.662,A 0.000,B 0.000,C 90.000,E1 119.127} C_DIS
LIN {X 0.151,Y -357.428,Z 1658.647,A 0.000,B 0.000,C 90.000,E1 116.360} C_DIS
LIN {X 0.048,Y -371.410,Z 1658.632,A 0.000,B 0.000,C 90.000,E1 113.695} C_DIS
LIN {X 0.106,Y -385.185,Z 1658.619,A 0.000,B 0.000,C 90.000,E1 111.354} C_DIS
LIN {X 0.013,Y -400.329,Z 1658.606,A 0.000,B 0.000,C 90.000,E1 109.087} C_DIS
LIN {X 0.025,Y -416.944,Z 1658.594,A 0.000,B 0.000,C 90.000,E1 106.858} C_DIS
LIN {X -0.203,Y -435.146,Z 1658.582,A 0.000,B 0.000,C 90.000,E1 104.717} C_DIS
LIN {X 0.098,Y -454.807,Z 1658.570,A 0.000,B 0.000,C 90.000,E1 102.591} C_DIS
LIN {X 0.175,Y -475.104,Z 1658.559,A 0.000,B 0.000,C 90.000,E1 100.658} C_DIS
LIN {X -0.187,Y -501.041,Z 1658.547,A 0.000,B 0.000,C 90.000,E1 98.511} C_DIS
LIN {X 0.072,Y -504.529,Z 1658.545,A 0.000,B 0.000,C 90.000,E1 98.049} C_DIS
LIN {X 0.003,Y -505.823,Z 1658.543,A 0.000,B 0.000,C 90.000,E1 97.814} C_DIS
LIN {X -0.135,Y -506.768,Z 1658.542,A 0.000,B 0.000,C 90.000,E1 97.587} C_DIS
LIN {X 0.187,Y -507.783,Z 1658.539,A 0.000,B 0.000,C 90.000,E1 97.068} C_DIS
LIN {X 0.012,Y -507.772,Z 1658.537,A 0.000,B 0.000,C 90.000,E1 96.606} C_DIS
LIN {X -0.157,Y -506.733,Z 1658.534,A 0.000,B 0.000,C 90.000,E1 96.144} C_DIS
LIN {X -0.217,Y -505.778,Z 1658.533,A 0.000,B 0.000,C 90.000,E1 95.910} C_DIS
LIN {X 0.175,Y -504.472,Z 1658.531,A 0.000,B 0.000,C 90.000,E1 95.625} C_DIS
LIN {X -0.069,Y -492.351,Z 1658.522,A 0.000,B 0.000,C 90.000,E1 93.955} C_DIS
LIN {X -0.114,Y -480.143,Z 1658.512,A 0.000,B 0.000,C 90.000,E1 92.236} C_DIS
LIN {X -0.201,Y -469.419,Z 1658.504,A 0.000,B 0.000,C 90.000,E1 90.745} C_DIS
LIN {X 0.223,Y -456.736,Z 1658.494,A 0.000,B 0.000,C 90.000,E1 88.912} C_DIS
LIN {X -0.009,Y -447.489,Z 1658.487,A 0.000,B 0.000,C 90.000,E1 87.650} C_DIS
LIN {X 0.071,Y -437.865,Z 1658.480,A 0.000,B 0.000,C 90.000,E1 86.331} C_DIS
LIN {X -0.082,Y -424.315,Z 1658.469,A 0.000,B 0.000,C 90.000,E1 84.489} C_DIS
LIN {X -0.201,Y -405.281,Z 1658.454,A 0.000,B 0.000,C 90.000,E1 81.781} C_DIS
LIN {X 0.155,Y -387.453,Z 1658.439,A 0.000,B 0.000,C 90.000,E1 78.926} C_DIS
LIN {X 0.039,Y -373.856,Z 1658.426,A 0.000,B 0.000,C 90.000,E1 76.645} C_DIS
LIN {X 0.125,Y -360.690,Z 1658.413,A 0.000,B 0.000,C 90.000,E1 74.283} C_DIS
LIN {X 0.106,Y -346.484,Z 1658.398,A 0.000,B 0.000,C 90.000,E1 71.583} C_DIS
LIN {X -0.063,Y -333.122,Z 1658.382,A 0.000,B 0.000,C 90.000,E1 68.847} C_DIS
LIN {X 0.146,Y -319.012,Z 1658.365,A 0.000,B 0.000,C 90.000,E1 65.665} C_DIS
LIN {X -0.040,Y -308.152,Z 1658.351,A 0.000,B 0.000,C 90.000,E1 63.127} C_DIS
LIN {X -0.085,Y -298.695,Z 1658.338,A 0.000,B 0.000,C 90.000,E1 60.845} C_DIS
LIN {X 0.070,Y -290.389,Z 1658.327,A 0.000,B 0.000,C 90.000,E1 58.820} C_DIS
LIN {X -0.127,Y -281.825,Z 1658.316,A 0.000,B 0.000,C 90.000,E1 56.834} C_DIS
LIN {X 0.009,Y -271.655,Z 1658.302,A 0.000,B 0.000,C 90.000,E1 54.402} C_DIS
LIN {X -0.144,Y -261.737,Z 1658.289,A 0.000,B 0.000,C 90.000,E1 51.984} C_DIS
LIN {X 0.024,Y -249.699,Z 1658.271,A 0.000,B 0.000,C 90.000,E1 48.728} C_DIS
LIN {X 0.133,Y -238.597,Z 1658.252,A 0.000,B 0.000,C 90.000,E1 45.405} C_DIS
LIN {X -0.050,Y -228.230,Z 1658.234,A 0.000,B 0.000,C 90.000,E1 42.081} C_DIS
LIN {X -0.070,Y -219.708,Z 1658.217,A 0.000,B 0.000,C 90.000,E1 39.036} C_DIS
LIN {X -0.057,Y -211.859,Z 1658.200,A 0.000,B 0.000,C 90.000,E1 35.931} C_DIS
LIN {X 0.030,Y -204.626,Z 1658.182,A 0.000,B 0.000,C 90.000,E1 32.752} C_DIS
LIN {X 0.065,Y -198.002,Z 1658.164,A 0.000,B 0.000,C 90.000,E1 29.539} C_DIS
LIN {X -0.003,Y -192.008,Z 1658.146,A 0.000,B 0.000,C 90.000,E1 26.309} C_DIS
LIN {X -0.034,Y -186.686,Z 1658.128,A 0.000,B 0.000,C 90.000,E1 23.025} C_DIS
LIN {X -0.005,Y -182.029,Z 1658.109,A 0.000,B 0.000,C 90.000,E1 19.685} C_DIS
LIN {X 0.003,Y -178.125,Z 1658.091,A 0.000,B 0.000,C 90.000,E1 16.315} C_DIS
LIN {X 0.010,Y -174.142,Z 1658.067,A 0.000,B 0.000,C 90.000,E1 12.063} C_DIS
LIN {X 0.061,Y -171.072,Z 1658.043,A 0.000,B 0.000,C 90.000,E1 7.757} C_DIS
LIN {X 0.045,Y -168.514,Z 1658.014,A 0.000,B 0.000,C 90.000,E1 2.579} C_DIS
LIN {X -0.017,Y -167.151,Z 1657.968,A 0.000,B 0.000,C 90.000,E1 354.318} C_DIS
LIN {X 0.059,Y -168.876,Z 1657.925,A 0.000,B 0.000,C 90.000,E1 346.464} C_DIS
LIN {X 0.047,Y -171.989,Z 1657.896,A 0.000,B 0.000,C 90.000,E1 341.275} C_DIS
LIN {X 0.064,Y -175.959,Z 1657.872,A 0.000,B 0.000,C 90.000,E1 336.975} C_DIS
LIN {X 0.000,Y -180.079,Z 1657.853,A 0.000,B 0.000,C 90.000,E1 333.589} C_DIS
LIN {X 0.032,Y -185.010,Z 1657.834,A 0.000,B 0.000,C 90.000,E1 330.205} C_DIS
LIN {X -0.111,Y -190.744,Z 1657.816,A 0.000,B 0.000,C 90.000,E1 326.914} C_DIS
LIN {X 0.043,Y -197.578,Z 1657.798,A 0.000,B 0.000,C 90.000,E1 323.577} C_DIS
LIN {X 0.106,Y -204.388,Z 1657.782,A 0.000,B 0.000,C 90.000,E1 320.723} C_DIS
LIN {X 0.019,Y -212.084,Z 1657.766,A 0.000,B 0.000,C 90.000,E1 317.957} C_DIS
LIN {X -0.087,Y -220.680,Z 1657.751,A 0.000,B 0.000,C 90.000,E1 315.243} C_DIS
LIN {X -0.052,Y -231.821,Z 1657.734,A 0.000,B 0.000,C 90.000,E1 312.162} C_DIS
LIN {X 0.024,Y -241.045,Z 1657.722,A 0.000,B 0.000,C 90.000,E1 309.886} C_DIS
LIN {X -0.026,Y -251.287,Z 1657.709,A 0.000,B 0.000,C 90.000,E1 307.684} C_DIS
LIN {X 0.002,Y -264.781,Z 1657.695,A 0.000,B 0.000,C 90.000,E1 305.152} C_DIS
LIN {X 0.042,Y -281.928,Z 1657.680,A 0.000,B 0.000,C 90.000,E1 302.339} C_DIS
LIN {X -0.161,Y -298.335,Z 1657.667,A 0.000,B 0.000,C 90.000,E1 300.001} C_DIS
LIN {X 0.022,Y -318.315,Z 1657.652,A 0.000,B 0.000,C 90.000,E1 297.334} C_DIS
LIN {X 0.114,Y -330.623,Z 1657.643,A 0.000,B 0.000,C 90.000,E1 295.720} C_DIS
LIN {X -0.187,Y -342.808,Z 1657.634,A 0.000,B 0.000,C 90.000,E1 294.207} C_DIS
LIN {X 0.003,Y -355.031,Z 1657.626,A 0.000,B 0.000,C 90.000,E1 292.642} C_DIS
LIN {X -0.074,Y -367.061,Z 1657.617,A 0.000,B 0.000,C 90.000,E1 291.153} C_DIS
LIN {X 0.039,Y -374.099,Z 1657.613,A 0.000,B 0.000,C 90.000,E1 290.248} C_DIS
LIN {X -0.124,Y -380.699,Z 1657.608,A 0.000,B 0.000,C 90.000,E1 289.396} C_DIS
LIN {X 0.129,Y -386.788,Z 1657.603,A 0.000,B 0.000,C 90.000,E1 288.489} C_DIS
LIN {X 0.079,Y -392.163,Z 1657.598,A 0.000,B 0.000,C 90.000,E1 287.638} C_DIS
LIN {X -0.047,Y -396.760,Z 1657.593,A 0.000,B 0.000,C 90.000,E1 286.804} C_DIS
LIN {X -0.195,Y -399.341,Z 1657.590,A 0.000,B 0.000,C 90.000,E1 286.260} C_DIS
LIN {X 0.055,Y -401.510,Z 1657.587,A 0.000,B 0.000,C 90.000,E1 285.662} C_DIS
LIN {X -0.173,Y -403.335,Z 1657.584,A 0.000,B 0.000,C 90.000,E1 285.134} C_DIS
LIN {X 0.099,Y -404.797,Z 1657.581,A 0.000,B 0.000,C 90.000,E1 284.537} C_DIS
LIN {X -0.110,Y -405.825,Z 1657.578,A 0.000,B 0.000,C 90.000,E1 284.008} C_DIS
LIN {X 0.180,Y -406.442,Z 1657.575,A 0.000,B 0.000,C 90.000,E1 283.411} C_DIS
LIN {X -0.015,Y -406.674,Z 1657.572,A 0.000,B 0.000,C 90.000,E1 282.883} C_DIS
LIN {X 0.191,Y -406.367,Z 1657.568,A 0.000,B 0.000,C 90.000,E1 282.299} C_DIS
LIN {X 0.002,Y -405.567,Z 1657.565,A 0.000,B 0.000,C 90.000,E1 281.771} C_DIS
LIN {X -0.188,Y -404.267,Z 1657.562,A 0.000,B 0.000,C 90.000,E1 281.243} C_DIS
LIN {X 0.011,Y -402.408,Z 1657.559,A 0.000,B 0.000,C 90.000,E1 280.658} C_DIS
LIN {X 0.130,Y -399.957,Z 1657.556,A 0.000,B 0.000,C 90.000,E1 280.084} C_DIS
LIN {X -0.090,Y -396.851,Z 1657.553,A 0.000,B 0.000,C 90.000,E1 279.557} C_DIS
LIN {X 0.067,Y -391.152,Z 1657.548,A 0.000,B 0.000,C 90.000,E1 278.690} C_DIS
LIN {X -0.149,Y -384.792,Z 1657.544,A 0.000,B 0.000,C 90.000,E1 277.871} C_DIS
LIN {X -0.103,Y -377.543,Z 1657.539,A 0.000,B 0.000,C 90.000,E1 277.004} C_DIS
LIN {X -0.044,Y -372.174,Z 1657.536,A 0.000,B 0.000,C 90.000,E1 276.429} C_DIS
LIN {X -0.167,Y -366.367,Z 1657.533,A 0.000,B 0.000,C 90.000,E1 275.910} C_DIS
LIN {X -0.013,Y -360.197,Z 1657.530,A 0.000,B 0.000,C 90.000,E1 275.391} C_DIS
LIN {X 0.076,Y -353.823,Z 1657.527,A 0.000,B 0.000,C 90.000,E1 274.935} C_DIS
LIN {X 0.046,Y -344.136,Z 1657.524,A 0.000,B 0.000,C 90.000,E1 274.359} C_DIS
LIN {X 0.076,Y -334.746,Z 1657.521,A 0.000,B 0.000,C 90.000,E1 273.841} C_DIS
LIN {X -0.060,Y -325.030,Z 1657.519,A 0.000,B 0.000,C 90.000,E1 273.383} C_DIS
LIN {X 0.110,Y -315.059,Z 1657.516,A 0.000,B 0.000,C 90.000,E1 272.922} C_DIS
LIN {X -0.096,Y -304.742,Z 1657.514,A 0.000,B 0.000,C 90.000,E1 272.579} C_DIS
LIN {X -0.037,Y -297.613,Z 1657.513,A 0.000,B 0.000,C 90.000,E1 272.350} C_DIS
LIN {X -0.133,Y -289.942,Z 1657.512,A 0.000,B 0.000,C 90.000,E1 272.178} C_DIS
LIN {X -0.060,Y -281.677,Z 1657.511,A 0.000,B 0.000,C 90.000,E1 272.007} C_DIS
LIN {X -0.121,Y -271.740,Z 1657.510,A 0.000,B 0.000,C 90.000,E1 271.892} C_DIS
LIN {X -0.078,Y -236.114,Z 1657.509,A 0.000,B 0.000,C 90.000,E1 271.661} C_DIS
LIN {X -0.018,Y -191.421,Z 1657.508,A 0.000,B 0.000,C 90.000,E1 271.432} C_DIS
LIN {X -0.058,Y -187.962,Z 1657.508,A 0.000,B 0.000,C 90.000,E1 271.432} C_DIS
LIN {X -0.085,Y -181.370,Z 1657.508,A 0.000,B 0.000,C 90.000,E1 271.432} C_DIS
LIN {X -0.058,Y -181.566,Z 1657.503,A 0.000,B 0.000,C 90.000,E1 270.516} C_DIS
LIN {X -0.069,Y -181.119,Z 1657.489,A 0.000,B 0.000,C 90.000,E1 267.993} C_DIS
LIN {X -0.080,Y -180.907,Z 1657.475,A 0.000,B 0.000,C 90.000,E1 265.469} C_DIS
LIN {X -0.023,Y -180.725,Z 1657.470,A 0.000,B 0.000,C 90.000,E1 264.609} C_DIS
LIN {X 0.075,Y -178.814,Z 1657.442,A 0.000,B 0.000,C 90.000,E1 259.511} C_DIS
LIN {X -0.019,Y -175.858,Z 1657.414,A 0.000,B 0.000,C 90.000,E1 254.448} C_DIS
LIN {X -0.036,Y -173.187,Z 1657.395,A 0.000,B 0.000,C 90.000,E1 251.040} C_DIS
LIN {X -0.035,Y -171.489,Z 1657.380,A 0.000,B 0.000,C 90.000,E1 248.465} C_DIS
LIN {X -0.047,Y -167.719,Z 1657.356,A 0.000,B 0.000,C 90.000,E1 244.152} C_DIS
LIN {X -0.031,Y -166.410,Z 1657.347,A 0.000,B 0.000,C 90.000,E1 242.410} C_DIS
LIN {X -0.032,Y -163.133,Z 1657.327,A 0.000,B 0.000,C 90.000,E1 238.918} C_DIS
LIN {X -0.067,Y -161.086,Z 1657.313,A 0.000,B 0.000,C 90.000,E1 236.294} C_DIS
LIN {X 0.043,Y -157.816,Z 1657.293,A 0.000,B 0.000,C 90.000,E1 232.718} C_DIS
LIN {X -0.019,Y -155.850,Z 1657.278,A 0.000,B 0.000,C 90.000,E1 230.070} C_DIS
LIN {X 0.037,Y -152.101,Z 1657.253,A 0.000,B 0.000,C 90.000,E1 225.567} C_DIS
LIN {X 0.056,Y -150.352,Z 1657.238,A 0.000,B 0.000,C 90.000,E1 222.852} C_DIS
LIN {X -0.015,Y -147.088,Z 1657.213,A 0.000,B 0.000,C 90.000,E1 218.338} C_DIS
LIN {X -0.020,Y -145.659,Z 1657.198,A 0.000,B 0.000,C 90.000,E1 215.598} C_DIS
LIN {X -0.017,Y -143.041,Z 1657.172,A 0.000,B 0.000,C 90.000,E1 211.003} C_DIS
LIN {X -0.016,Y -141.666,Z 1657.152,A 0.000,B 0.000,C 90.000,E1 207.308} C_DIS
LIN {X 0.028,Y -139.450,Z 1657.116,A 0.000,B 0.000,C 90.000,E1 200.791} C_DIS
LIN {X -0.051,Y -139.184,Z 1657.105,A 0.000,B 0.000,C 90.000,E1 198.960} C_DIS
LIN {X -0.028,Y -138.322,Z 1657.053,A 0.000,B 0.000,C 90.000,E1 189.613} C_DIS
LIN {X -0.021,Y -139.462,Z 1657.007,A 0.000,B 0.000,C 90.000,E1 181.203} C_DIS
LIN {X 0.060,Y -141.021,Z 1656.976,A 0.000,B 0.000,C 90.000,E1 175.584} C_DIS
LIN {X 0.014,Y -142.384,Z 1656.960,A 0.000,B 0.000,C 90.000,E1 172.818} C_DIS
LIN {X -0.064,Y -144.615,Z 1656.934,A 0.000,B 0.000,C 90.000,E1 168.229} C_DIS
LIN {X -0.003,Y -147.810,Z 1656.909,A 0.000,B 0.000,C 90.000,E1 163.614} C_DIS
LIN {X 0.084,Y -150.497,Z 1656.889,A 0.000,B 0.000,C 90.000,E1 159.934} C_DIS
LIN {X -0.035,Y -153.955,Z 1656.869,A 0.000,B 0.000,C 90.000,E1 156.357} C_DIS
LIN {X 0.027,Y -157.366,Z 1656.849,A 0.000,B 0.000,C 90.000,E1 152.743} C_DIS
LIN {X -0.030,Y -161.566,Z 1656.829,A 0.000,B 0.000,C 90.000,E1 149.203} C_DIS
LIN {X -0.019,Y -165.764,Z 1656.809,A 0.000,B 0.000,C 90.000,E1 145.674} C_DIS
LIN {X -0.032,Y -170.720,Z 1656.790,A 0.000,B 0.000,C 90.000,E1 142.190} C_DIS
LIN {X 0.010,Y -175.593,Z 1656.771,A 0.000,B 0.000,C 90.000,E1 138.728} C_DIS
LIN {X -0.003,Y -181.210,Z 1656.752,A 0.000,B 0.000,C 90.000,E1 135.324} C_DIS
LIN {X -0.011,Y -186.675,Z 1656.733,A 0.000,B 0.000,C 90.000,E1 131.962} C_DIS
LIN {X -0.066,Y -191.277,Z 1656.719,A 0.000,B 0.000,C 90.000,E1 129.483} C_DIS
LIN {X 0.014,Y -197.102,Z 1656.701,A 0.000,B 0.000,C 90.000,E1 126.171} C_DIS
LIN {X 0.050,Y -200.377,Z 1656.692,A 0.000,B 0.000,C 90.000,E1 124.532} C_DIS
LIN {X 0.013,Y -207.206,Z 1656.671,A 0.000,B 0.000,C 90.000,E1 120.846} C_DIS
LIN {X -0.028,Y -327.861,Z 1656.671,A 0.000,B 0.000,C 90.000,E1 120.846} C_DIS
LIN {X 0.110,Y -329.745,Z 1656.671,A 0.000,B 0.000,C 90.000,E1 120.797} C_DIS
LIN {X -0.097,Y -335.723,Z 1656.670,A 0.000,B 0.000,C 90.000,E1 120.541} C_DIS
LIN {X 0.103,Y -338.822,Z 1656.668,A 0.000,B 0.000,C 90.000,E1 120.207} C_DIS
LIN {X 0.116,Y -342.408,Z 1656.665,A 0.000,B 0.000,C 90.000,E1 119.667} C_DIS
LIN {X 0.165,Y -351.930,Z 1656.653,A 0.000,B 0.000,C 90.000,E1 117.513} C_DIS
LIN {X 0.065,Y -365.264,Z 1656.638,A 0.000,B 0.000,C 90.000,E1 114.823} C_DIS
LIN {X -0.125,Y -380.152,Z 1656.623,A 0.000,B 0.000,C 90.000,E1 112.206} C_DIS
LIN {X 0.016,Y -394.802,Z 1656.610,A 0.000,B 0.000,C 90.000,E1 109.885} C_DIS
LIN {X 0.023,Y -410.885,Z 1656.598,A 0.000,B 0.000,C 90.000,E1 107.638} C_DIS
LIN {X 0.177,Y -428.513,Z 1656.586,A 0.000,B 0.000,C 90.000,E1 105.426} C_DIS
LIN {X 0.178,Y -447.747,Z 1656.574,A 0.000,B 0.000,C 90.000,E1 103.300} C_DIS
LIN {X -0.212,Y -467.850,Z 1656.563,A 0.000,B 0.000,C 90.000,E1 101.366} C_DIS
LIN {X -0.189,Y -491.110,Z 1656.552,A 0.000,B 0.000,C 90.000,E1 99.321} C_DIS
LIN {X -0.170,Y -498.978,Z 1656.548,A 0.000,B 0.000,C 90.000,E1 98.681} C_DIS
LIN {X -0.023,Y -501.361,Z 1656.547,A 0.000,B 0.000,C 90.000,E1 98.454} C_DIS
LIN {X 0.080,Y -503.264,Z 1656.546,A 0.000,B 0.000,C 90.000,E1 98.219} C_DIS
LIN {X 0.111,Y -504.716,Z 1656.544,A 0.000,B 0.000,C 90.000,E1 97.992} C_DIS
LIN {X 0.049,Y -505.905,Z 1656.543,A 0.000,B 0.000,C 90.000,E1 97.757} C_DIS
LIN {X -0.083,Y -506.764,Z 1656.542,A 0.000,B 0.000,C 90.000,E1 97.530} C_DIS
LIN {X -0.263,Y -507.637,Z 1656.539,A 0.000,B 0.000,C 90.000,E1 97.068} C_DIS
LIN {X 0.066,Y -507.494,Z 1656.536,A 0.000,B 0.000,C 90.000,E1 96.549} C_DIS
LIN {X -0.104,Y -506.311,Z 1656.534,A 0.000,B 0.000,C 90.000,E1 96.087} C_DIS
LIN {X -0.163,Y -505.269,Z 1656.532,A 0.000,B 0.000,C 90.000,E1 95.853} C_DIS
LIN {X 0.227,Y -503.858,Z 1656.531,A 0.000,B 0.000,C 90.000,E1 95.568} C_DIS
LIN {X 0.074,Y -493.471,Z 1656.523,A 0.000,B 0.000,C 90.000,E1 94.131} C_DIS
LIN {X 0.074,Y -481.284,Z 1656.513,A 0.000,B 0.000,C 90.000,E1 92.407} C_DIS
LIN {X 0.001,Y -470.620,Z 1656.505,A 0.000,B 0.000,C 90.000,E1 90.917} C_DIS
LIN {X -0.007,Y -457.952,Z 1656.495,A 0.000,B 0.000,C 90.000,E1 89.141} C_DIS
LIN {X -0.013,Y -446.837,Z 1656.487,A 0.000,B 0.000,C 90.000,E1 87.593} C_DIS
LIN {X 0.057,Y -437.185,Z 1656.479,A 0.000,B 0.000,C 90.000,E1 86.274} C_DIS
LIN {X -0.110,Y -423.617,Z 1656.469,A 0.000,B 0.000,C 90.000,E1 84.432} C_DIS
LIN {X 0.209,Y -404.588,Z 1656.454,A 0.000,B 0.000,C 90.000,E1 81.659} C_DIS
LIN {X 0.083,Y -386.778,Z 1656.438,A 0.000,B 0.000,C 90.000,E1 78.870} C_DIS
LIN {X -0.048,Y -373.185,Z 1656.425,A 0.000,B 0.000,C 90.000,E1 76.589} C_DIS
LIN {X 0.078,Y -358.445,Z 1656.411,A 0.000,B 0.000,C 90.000,E1 73.921} C_DIS
LIN {X 0.025,Y -342.837,Z 1656.394,A 0.000,B 0.000,C 90.000,E1 70.913} C_DIS
LIN {X -0.098,Y -331.059,Z 1656.380,A 0.000,B 0.000,C 90.000,E1 68.465} C_DIS
LIN {X 0.059,Y -317.038,Z 1656.363,A 0.000,B 0.000,C 90.000,E1 65.281} C_DIS
LIN {X -0.073,Y -307.580,Z 1656.350,A 0.000,B 0.000,C 90.000,E1 63.050} C_DIS
LIN {X 0.119,Y -299.478,Z 1656.339,A 0.000,B 0.000,C 90.000,E1 61.051} C_DIS
LIN {X 0.032,Y -291.182,Z 1656.328,A 0.000,B 0.000,C 90.000,E1 59.076} C_DIS
LIN {X 0.115,Y -284.110,Z 1656.319,A 0.000,B 0.000,C 90.000,E1 57.375} C_DIS
LIN {X 0.037,Y -275.410,Z 1656.307,A 0.000,B 0.000,C 90.000,E1 55.341} C_DIS
LIN {X 0.030,Y -264.023,Z 1656.292,A 0.000,B 0.000,C 90.000,E1 52.557} C_DIS
LIN {X -0.097,Y -251.812,Z 1656.274,A 0.000,B 0.000,C 90.000,E1 49.380} C_DIS
LIN {X 0.092,Y -240.516,Z 1656.256,A 0.000,B 0.000,C 90.000,E1 46.053} C_DIS
LIN {X 0.004,Y -231.170,Z 1656.239,A 0.000,B 0.000,C 90.000,E1 43.095} C_DIS
LIN {X -0.063,Y -223.415,Z 1656.225,A 0.000,B 0.000,C 90.000,E1 40.458} C_DIS
LIN {X 0.006,Y -215.218,Z 1656.208,A 0.000,B 0.000,C 90.000,E1 37.363} C_DIS
LIN {X -0.049,Y -207.723,Z 1656.190,A 0.000,B 0.000,C 90.000,E1 34.246} C_DIS
LIN {X -0.006,Y -200.841,Z 1656.172,A 0.000,B 0.000,C 90.000,E1 31.052} C_DIS
LIN {X -0.088,Y -194.569,Z 1656.155,A 0.000,B 0.000,C 90.000,E1 27.847} C_DIS
LIN {X 0.103,Y -188.934,Z 1656.136,A 0.000,B 0.000,C 90.000,E1 24.515} C_DIS
LIN {X 0.013,Y -184.026,Z 1656.118,A 0.000,B 0.000,C 90.000,E1 21.227} C_DIS
LIN {X 0.019,Y -179.813,Z 1656.099,A 0.000,B 0.000,C 90.000,E1 17.873} C_DIS
LIN {X -0.007,Y -175.512,Z 1656.076,A 0.000,B 0.000,C 90.000,E1 13.647} C_DIS
LIN {X -0.022,Y -172.127,Z 1656.052,A 0.000,B 0.000,C 90.000,E1 9.378} C_DIS
LIN {X 0.032,Y -169.190,Z 1656.023,A 0.000,B 0.000,C 90.000,E1 4.188} C_DIS
LIN {X 0.011,Y -167.199,Z 1655.973,A 0.000,B 0.000,C 90.000,E1 355.179} C_DIS
LIN {X 0.062,Y -168.930,Z 1655.925,A 0.000,B 0.000,C 90.000,E1 346.464} C_DIS
LIN {X 0.053,Y -172.066,Z 1655.896,A 0.000,B 0.000,C 90.000,E1 341.275} C_DIS
LIN {X 0.073,Y -176.051,Z 1655.872,A 0.000,B 0.000,C 90.000,E1 336.975} C_DIS
LIN {X 0.012,Y -180.192,Z 1655.853,A 0.000,B 0.000,C 90.000,E1 333.589} C_DIS
LIN {X 0.046,Y -185.154,Z 1655.835,A 0.000,B 0.000,C 90.000,E1 330.205} C_DIS
LIN {X -0.093,Y -190.919,Z 1655.816,A 0.000,B 0.000,C 90.000,E1 326.914} C_DIS
LIN {X -0.093,Y -197.748,Z 1655.798,A 0.000,B 0.000,C 90.000,E1 323.623} C_DIS
LIN {X 0.005,Y -204.567,Z 1655.782,A 0.000,B 0.000,C 90.000,E1 320.759} C_DIS
LIN {X 0.052,Y -212.248,Z 1655.766,A 0.000,B 0.000,C 90.000,E1 317.957} C_DIS
LIN {X -0.049,Y -220.841,Z 1655.751,A 0.000,B 0.000,C 90.000,E1 315.243} C_DIS
LIN {X 0.044,Y -230.501,Z 1655.736,A 0.000,B 0.000,C 90.000,E1 312.528} C_DIS
LIN {X 0.072,Y -241.161,Z 1655.722,A 0.000,B 0.000,C 90.000,E1 309.886} C_DIS
LIN {X 0.025,Y -251.378,Z 1655.709,A 0.000,B 0.000,C 90.000,E1 307.684} C_DIS
LIN {X 0.059,Y -264.846,Z 1655.695,A 0.000,B 0.000,C 90.000,E1 305.152} C_DIS
LIN {X 0.013,Y -279.712,Z 1655.682,A 0.000,B 0.000,C 90.000,E1 302.704} C_DIS
LIN {X -0.094,Y -298.369,Z 1655.667,A 0.000,B 0.000,C 90.000,E1 300.001} C_DIS
LIN {X 0.095,Y -318.345,Z 1655.652,A 0.000,B 0.000,C 90.000,E1 297.334} C_DIS
LIN {X 0.190,Y -330.656,Z 1655.643,A 0.000,B 0.000,C 90.000,E1 295.720} C_DIS
LIN {X -0.108,Y -342.804,Z 1655.634,A 0.000,B 0.000,C 90.000,E1 294.207} C_DIS
LIN {X 0.085,Y -355.001,Z 1655.626,A 0.000,B 0.000,C 90.000,E1 292.642} C_DIS
LIN {X 0.010,Y -367.034,Z 1655.618,A 0.000,B 0.000,C 90.000,E1 291.153} C_DIS
LIN {X 0.124,Y -374.073,Z 1655.613,A 0.000,B 0.000,C 90.000,E1 290.248} C_DIS
LIN {X -0.038,Y -380.675,Z 1655.608,A 0.000,B 0.000,C 90.000,E1 289.396} C_DIS
LIN {X -0.150,Y -386.743,Z 1655.603,A 0.000,B 0.000,C 90.000,E1 288.544} C_DIS
LIN {X 0.168,Y -392.167,Z 1655.598,A 0.000,B 0.000,C 90.000,E1 287.638} C_DIS
LIN {X -0.007,Y -395.354,Z 1655.595,A 0.000,B 0.000,C 90.000,E1 287.094} C_DIS
LIN {X 0.217,Y -398.154,Z 1655.592,A 0.000,B 0.000,C 90.000,E1 286.496} C_DIS
LIN {X 0.147,Y -401.593,Z 1655.587,A 0.000,B 0.000,C 90.000,E1 285.662} C_DIS
LIN {X -0.081,Y -403.413,Z 1655.584,A 0.000,B 0.000,C 90.000,E1 285.134} C_DIS
LIN {X 0.192,Y -404.897,Z 1655.581,A 0.000,B 0.000,C 90.000,E1 284.537} C_DIS
LIN {X -0.016,Y -405.920,Z 1655.578,A 0.000,B 0.000,C 90.000,E1 284.008} C_DIS
LIN {X -0.121,Y -406.616,Z 1655.575,A 0.000,B 0.000,C 90.000,E1 283.467} C_DIS
LIN {X 0.080,Y -406.818,Z 1655.572,A 0.000,B 0.000,C 90.000,E1 282.883} C_DIS
LIN {X -0.111,Y -406.520,Z 1655.569,A 0.000,B 0.000,C 90.000,E1 282.355} C_DIS
LIN {X 0.099,Y -405.763,Z 1655.565,A 0.000,B 0.000,C 90.000,E1 281.771} C_DIS
LIN {X -0.092,Y -404.462,Z 1655.562,A 0.000,B 0.000,C 90.000,E1 281.243} C_DIS
LIN {X 0.109,Y -402.591,Z 1655.559,A 0.000,B 0.000,C 90.000,E1 280.658} C_DIS
LIN {X -0.165,Y -400.106,Z 1655.556,A 0.000,B 0.000,C 90.000,E1 280.141} C_DIS
LIN {X 0.009,Y -397.007,Z 1655.553,A 0.000,B 0.000,C 90.000,E1 279.557} C_DIS
LIN {X 0.166,Y -391.292,Z 1655.548,A 0.000,B 0.000,C 90.000,E1 278.690} C_DIS
LIN {X -0.051,Y -384.906,Z 1655.544,A 0.000,B 0.000,C 90.000,E1 277.871} C_DIS
LIN {X -0.005,Y -377.681,Z 1655.539,A 0.000,B 0.000,C 90.000,E1 277.004} C_DIS
LIN {X 0.035,Y -372.216,Z 1655.536,A 0.000,B 0.000,C 90.000,E1 276.429} C_DIS
LIN {X -0.112,Y -366.333,Z 1655.533,A 0.000,B 0.000,C 90.000,E1 275.910} C_DIS
LIN {X 0.051,Y -360.155,Z 1655.530,A 0.000,B 0.000,C 90.000,E1 275.391} C_DIS
LIN {X 0.141,Y -353.755,Z 1655.528,A 0.000,B 0.000,C 90.000,E1 274.935} C_DIS
LIN {X 0.076,Y -343.981,Z 1655.524,A 0.000,B 0.000,C 90.000,E1 274.359} C_DIS
LIN {X 0.111,Y -334.603,Z 1655.521,A 0.000,B 0.000,C 90.000,E1 273.841} C_DIS
LIN {X -0.026,Y -324.905,Z 1655.519,A 0.000,B 0.000,C 90.000,E1 273.383} C_DIS
LIN {X 0.142,Y -314.878,Z 1655.516,A 0.000,B 0.000,C 90.000,E1 272.922} C_DIS
LIN {X -0.050,Y -304.486,Z 1655.514,A 0.000,B 0.000,C 90.000,E1 272.579} C_DIS
LIN {X 0.141,Y -293.712,Z 1655.513,A 0.000,B 0.000,C 90.000,E1 272.236} C_DIS
LIN {X -0.143,Y -286.136,Z 1655.512,A 0.000,B 0.000,C 90.000,E1 272.121} C_DIS
LIN {X 0.008,Y -277.554,Z 1655.511,A 0.000,B 0.000,C 90.000,E1 271.949} C_DIS
LIN {X 0.013,Y -265.203,Z 1655.510,A 0.000,B 0.000,C 90.000,E1 271.835} C_DIS
LIN {X -0.001,Y -236.933,Z 1655.509,A 0.000,B 0.000,C 90.000,E1 271.661} C_DIS
LIN {X -0.094,Y -197.487,Z 1655.508,A 0.000,B 0.000,C 90.000,E1 271.489} C_DIS
LIN {X -0.007,Y -187.586,Z 1655.508,A 0.000,B 0.000,C 90.000,E1 271.432} C_DIS
LIN {X -0.037,Y -181.367,Z 1655.508,A 0.000,B 0.000,C 90.000,E1 271.432} C_DIS
LIN {X 0.018,Y -181.563,Z 1655.503,A 0.000,B 0.000,C 90.000,E1 270.516} C_DIS
LIN {X -0.053,Y -181.283,Z 1655.494,A 0.000,B 0.000,C 90.000,E1 268.854} C_DIS
LIN {X -0.004,Y -180.907,Z 1655.475,A 0.000,B 0.000,C 90.000,E1 265.469} C_DIS
LIN {X 0.052,Y -180.736,Z 1655.470,A 0.000,B 0.000,C 90.000,E1 264.609} C_DIS
LIN {X -0.026,Y -178.826,Z 1655.442,A 0.000,B 0.000,C 90.000,E1 259.567} C_DIS
LIN {X 0.055,Y -175.870,Z 1655.414,A 0.000,B 0.000,C 90.000,E1 254.448} C_DIS
LIN {X 0.050,Y -173.841,Z 1655.400,A 0.000,B 0.000,C 90.000,E1 251.891} C_DIS
LIN {X 0.039,Y -171.510,Z 1655.380,A 0.000,B 0.000,C 90.000,E1 248.465} C_DIS
LIN {X 0.025,Y -167.737,Z 1655.356,A 0.000,B 0.000,C 90.000,E1 244.152} C_DIS
LIN {X 0.040,Y -166.435,Z 1655.347,A 0.000,B 0.000,C 90.000,E1 242.410} C_DIS
LIN {X -0.046,Y -163.154,Z 1655.327,A 0.000,B 0.000,C 90.000,E1 238.948} C_DIS
LIN {X 0.004,Y -161.111,Z 1655.313,A 0.000,B 0.000,C 90.000,E1 236.294} C_DIS
LIN {X -0.012,Y -157.837,Z 1655.293,A 0.000,B 0.000,C 90.000,E1 232.763} C_DIS
LIN {X 0.050,Y -155.869,Z 1655.278,A 0.000,B 0.000,C 90.000,E1 230.070} C_DIS
LIN {X -0.001,Y -152.119,Z 1655.253,A 0.000,B 0.000,C 90.000,E1 225.607} C_DIS
LIN {X 0.014,Y -150.370,Z 1655.238,A 0.000,B 0.000,C 90.000,E1 222.894} C_DIS
LIN {X -0.064,Y -147.104,Z 1655.213,A 0.000,B 0.000,C 90.000,E1 218.382} C_DIS
LIN {X 0.045,Y -145.672,Z 1655.198,A 0.000,B 0.000,C 90.000,E1 215.598} C_DIS
LIN {X 0.048,Y -143.054,Z 1655.172,A 0.000,B 0.000,C 90.000,E1 211.003} C_DIS
LIN {X -0.017,Y -141.676,Z 1655.152,A 0.000,B 0.000,C 90.000,E1 207.334} C_DIS
LIN {X -0.038,Y -139.455,Z 1655.116,A 0.000,B 0.000,C 90.000,E1 200.844} C_DIS
LIN {X 0.013,Y -139.189,Z 1655.105,A 0.000,B 0.000,C 90.000,E1 198.960} C_DIS
LIN {X 0.036,Y -138.323,Z 1655.053,A 0.000,B 0.000,C 90.000,E1 189.613} C_DIS
LIN {X 0.044,Y -139.458,Z 1655.007,A 0.000,B 0.000,C 90.000,E1 181.203} C_DIS
LIN {X -0.015,Y -141.010,Z 1654.976,A 0.000,B 0.000,C 90.000,E1 175.641} C_DIS
LIN {X -0.067,Y -142.764,Z 1654.955,A 0.000,B 0.000,C 90.000,E1 171.951} C_DIS
LIN {X 0.031,Y -145.170,Z 1654.929,A 0.000,B 0.000,C 90.000,E1 167.297} C_DIS
LIN {X 0.022,Y -147.793,Z 1654.909,A 0.000,B 0.000,C 90.000,E1 163.630} C_DIS
LIN {X -0.040,Y -150.475,Z 1654.889,A 0.000,B 0.000,C 90.000,E1 160.007} C_DIS
LIN {X 0.033,Y -153.929,Z 1654.869,A 0.000,B 0.000,C 90.000,E1 156.357} C_DIS
LIN {X -0.044,Y -157.340,Z 1654.849,A 0.000,B 0.000,C 90.000,E1 152.794} C_DIS
LIN {X 0.041,Y -161.533,Z 1654.829,A 0.000,B 0.000,C 90.000,E1 149.203} C_DIS
LIN {X 0.054,Y -165.732,Z 1654.809,A 0.000,B 0.000,C 90.000,E1 145.674} C_DIS
LIN {X 0.041,Y -170.682,Z 1654.790,A 0.000,B 0.000,C 90.000,E1 142.190} C_DIS
LIN {X -0.046,Y -175.556,Z 1654.771,A 0.000,B 0.000,C 90.000,E1 138.771} C_DIS
LIN {X 0.073,Y -181.175,Z 1654.752,A 0.000,B 0.000,C 90.000,E1 135.324} C_DIS
LIN {X -0.058,Y -186.633,Z 1654.733,A 0.000,B 0.000,C 90.000,E1 132.000} C_DIS
LIN {X 0.012,Y -191.239,Z 1654.719,A 0.000,B 0.000,C 90.000,E1 129.483} C_DIS
LIN {X -0.066,Y -197.057,Z 1654.701,A 0.000,B 0.000,C 90.000,E1 126.217} C_DIS
LIN {X 0.017,Y -200.329,Z 1654.692,A 0.000,B 0.000,C 90.000,E1 124.565} C_DIS
LIN {X 0.057,Y -207.122,Z 1654.672,A 0.000,B 0.000,C 90.000,E1 120.875} C_DIS
LIN {X 0.036,Y -327.567,Z 1654.672,A 0.000,B 0.000,C 90.000,E1 120.875} C_DIS
LIN {X -0.018,Y -328.618,Z 1654.672,A 0.000,B 0.000,C 90.000,E1 120.875} C_DIS
LIN {X -0.049,Y -333.357,Z 1654.671,A 0.000,B 0.000,C 90.000,E1 120.718} C_DIS
LIN {X 0.035,Y -335.748,Z 1654.670,A 0.000,B 0.000,C 90.000,E1 120.541} C_DIS
LIN {X 0.084,Y -339.602,Z 1654.667,A 0.000,B 0.000,C 90.000,E1 120.129} C_DIS
LIN {X -0.093,Y -341.493,Z 1654.666,A 0.000,B 0.000,C 90.000,E1 119.873} C_DIS
LIN {X -0.101,Y -342.980,Z 1654.664,A 0.000,B 0.000,C 90.000,E1 119.589} C_DIS
LIN {X -0.112,Y -356.716,Z 1654.647,A 0.000,B 0.000,C 90.000,E1 116.539} C_DIS
LIN {X 0.092,Y -370.615,Z 1654.632,A 0.000,B 0.000,C 90.000,E1 113.823} C_DIS
LIN {X -0.224,Y -384.314,Z 1654.620,A 0.000,B 0.000,C 90.000,E1 111.535} C_DIS
LIN {X 0.024,Y -399.377,Z 1654.607,A 0.000,B 0.000,C 90.000,E1 109.214} C_DIS
LIN {X 0.018,Y -415.904,Z 1654.594,A 0.000,B 0.000,C 90.000,E1 106.985} C_DIS
LIN {X -0.117,Y -434.012,Z 1654.582,A 0.000,B 0.000,C 90.000,E1 104.828} C_DIS
LIN {X 0.028,Y -453.601,Z 1654.571,A 0.000,B 0.000,C 90.000,E1 102.715} C_DIS
LIN {X 0.031,Y -473.868,Z 1654.560,A 0.000,B 0.000,C 90.000,E1 100.782} C_DIS
LIN {X -0.079,Y -497.289,Z 1654.549,A 0.000,B 0.000,C 90.000,E1 98.803} C_DIS
LIN {X 0.150,Y -499.885,Z 1654.548,A 0.000,B 0.000,C 90.000,E1 98.568} C_DIS
LIN {X -0.190,Y -501.985,Z 1654.547,A 0.000,B 0.000,C 90.000,E1 98.398} C_DIS
LIN {X -0.235,Y -503.802,Z 1654.545,A 0.000,B 0.000,C 90.000,E1 98.163} C_DIS
LIN {X 0.219,Y -505.164,Z 1654.544,A 0.000,B 0.000,C 90.000,E1 97.871} C_DIS
LIN {X 0.025,Y -506.886,Z 1654.541,A 0.000,B 0.000,C 90.000,E1 97.409} C_DIS
LIN {X -0.162,Y -507.496,Z 1654.538,A 0.000,B 0.000,C 90.000,E1 96.947} C_DIS
LIN {X 0.165,Y -507.097,Z 1654.536,A 0.000,B 0.000,C 90.000,E1 96.429} C_DIS
LIN {X -0.010,Y -505.625,Z 1654.533,A 0.000,B 0.000,C 90.000,E1 95.967} C_DIS
LIN {X -0.123,Y -504.405,Z 1654.532,A 0.000,B 0.000,C 90.000,E1 95.739} C_DIS
LIN {X -0.132,Y -495.905,Z 1654.525,A 0.000,B 0.000,C 90.000,E1 94.531} C_DIS
LIN {X -0.240,Y -481.995,Z 1654.514,A 0.000,B 0.000,C 90.000,E1 92.579} C_DIS
LIN {X 0.177,Y -471.397,Z 1654.506,A 0.000,B 0.000,C 90.000,E1 91.031} C_DIS
LIN {X -0.071,Y -460.550,Z 1654.497,A 0.000,B 0.000,C 90.000,E1 89.542} C_DIS
LIN {X -0.029,Y -449.505,Z 1654.489,A 0.000,B 0.000,C 90.000,E1 87.993} C_DIS
LIN {X 0.084,Y -439.942,Z 1654.482,A 0.000,B 0.000,C 90.000,E1 86.674} C_DIS
LIN {X 0.101,Y -424.395,Z 1654.470,A 0.000,B 0.000,C 90.000,E1 84.546} C_DIS
LIN {X -0.022,Y -405.300,Z 1654.455,A 0.000,B 0.000,C 90.000,E1 81.837} C_DIS
LIN {X -0.127,Y -387.411,Z 1654.439,A 0.000,B 0.000,C 90.000,E1 79.050} C_DIS
LIN {X 0.209,Y -373.800,Z 1654.426,A 0.000,B 0.000,C 90.000,E1 76.700} C_DIS
LIN {X -0.090,Y -359.040,Z 1654.412,A 0.000,B 0.000,C 90.000,E1 74.102} C_DIS
LIN {X -0.120,Y -343.372,Z 1654.395,A 0.000,B 0.000,C 90.000,E1 71.094} C_DIS
LIN {X 0.085,Y -331.563,Z 1654.381,A 0.000,B 0.000,C 90.000,E1 68.592} C_DIS
LIN {X -0.174,Y -317.482,Z 1654.364,A 0.000,B 0.000,C 90.000,E1 65.485} C_DIS
LIN {X -0.025,Y -308.030,Z 1654.351,A 0.000,B 0.000,C 90.000,E1 63.204} C_DIS
LIN {X -0.098,Y -299.941,Z 1654.340,A 0.000,B 0.000,C 90.000,E1 61.257} C_DIS
LIN {X -0.023,Y -291.691,Z 1654.329,A 0.000,B 0.000,C 90.000,E1 59.253} C_DIS
LIN {X -0.100,Y -283.196,Z 1654.318,A 0.000,B 0.000,C 90.000,E1 57.248} C_DIS
LIN {X -0.035,Y -274.484,Z 1654.307,A 0.000,B 0.000,C 90.000,E1 55.182} C_DIS
LIN {X -0.055,Y -263.158,Z 1654.291,A 0.000,B 0.000,C 90.000,E1 52.396} C_DIS
LIN {X -0.006,Y -251.027,Z 1654.273,A 0.000,B 0.000,C 90.000,E1 49.175} C_DIS
LIN {X -0.023,Y -239.802,Z 1654.255,A 0.000,B 0.000,C 90.000,E1 45.891} C_DIS
LIN {X -0.010,Y -229.287,Z 1654.236,A 0.000,B 0.000,C 90.000,E1 42.528} C_DIS
LIN {X -0.016,Y -220.602,Z 1654.219,A 0.000,B 0.000,C 90.000,E1 39.483} C_DIS
LIN {X 0.020,Y -212.605,Z 1654.202,A 0.000,B 0.000,C 90.000,E1 36.377} C_DIS
LIN {X -0.042,Y -205.285,Z 1654.185,A 0.000,B 0.000,C 90.000,E1 33.245} C_DIS
LIN {X -0.054,Y -198.618,Z 1654.167,A 0.000,B 0.000,C 90.000,E1 30.050} C_DIS
LIN {X -0.021,Y -192.592,Z 1654.149,A 0.000,B 0.000,C 90.000,E1 26.796} C_DIS
LIN {X -0.046,Y -187.225,Z 1654.131,A 0.000,B 0.000,C 90.000,E1 23.515} C_DIS
LIN {X -0.004,Y -182.547,Z 1654.112,A 0.000,B 0.000,C 90.000,E1 20.174} C_DIS
LIN {X 0.018,Y -178.614,Z 1654.093,A 0.000,B 0.000,C 90.000,E1 16.804} C_DIS
LIN {X -0.082,Y -174.601,Z 1654.070,A 0.000,B 0.000,C 90.000,E1 12.591} C_DIS
LIN {X 0.014,Y -171.449,Z 1654.046,A 0.000,B 0.000,C 90.000,E1 8.276} C_DIS
LIN {X 0.022,Y -168.797,Z 1654.017,A 0.000,B 0.000,C 90.000,E1 3.094} C_DIS
LIN {X -0.013,Y -167.238,Z 1653.968,A 0.000,B 0.000,C 90.000,E1 354.318} C_DIS
LIN {X 0.066,Y -169.002,Z 1653.925,A 0.000,B 0.000,C 90.000,E1 346.464} C_DIS
LIN {X 0.061,Y -172.145,Z 1653.896,A 0.000,B 0.000,C 90.000,E1 341.275} C_DIS
LIN {X 0.014,Y -176.155,Z 1653.872,A 0.000,B 0.000,C 90.000,E1 336.997} C_DIS
LIN {X 0.024,Y -180.320,Z 1653.853,A 0.000,B 0.000,C 90.000,E1 333.589} C_DIS
LIN {X 0.063,Y -185.299,Z 1653.835,A 0.000,B 0.000,C 90.000,E1 330.205} C_DIS
LIN {X -0.072,Y -191.092,Z 1653.816,A 0.000,B 0.000,C 90.000,E1 326.914} C_DIS
LIN {X -0.067,Y -197.928,Z 1653.798,A 0.000,B 0.000,C 90.000,E1 323.623} C_DIS
LIN {X 0.041,Y -205.773,Z 1653.780,A 0.000,B 0.000,C 90.000,E1 320.356} C_DIS
LIN {X -0.031,Y -213.596,Z 1653.764,A 0.000,B 0.000,C 90.000,E1 317.595} C_DIS
LIN {X -0.009,Y -221.003,Z 1653.751,A 0.000,B 0.000,C 90.000,E1 315.243} C_DIS
LIN {X 0.090,Y -230.646,Z 1653.736,A 0.000,B 0.000,C 90.000,E1 312.528} C_DIS
LIN {X -0.062,Y -241.272,Z 1653.722,A 0.000,B 0.000,C 90.000,E1 309.930} C_DIS
LIN {X -0.117,Y -251.467,Z 1653.709,A 0.000,B 0.000,C 90.000,E1 307.729} C_DIS
LIN {X 0.078,Y -262.891,Z 1653.697,A 0.000,B 0.000,C 90.000,E1 305.518} C_DIS
LIN {X -0.097,Y -277.542,Z 1653.684,A 0.000,B 0.000,C 90.000,E1 303.086} C_DIS
LIN {X -0.021,Y -296.012,Z 1653.668,A 0.000,B 0.000,C 90.000,E1 300.335} C_DIS
LIN {X -0.169,Y -315.864,Z 1653.654,A 0.000,B 0.000,C 90.000,E1 297.719} C_DIS
LIN {X -0.058,Y -325.796,Z 1653.647,A 0.000,B 0.000,C 90.000,E1 296.411} C_DIS
LIN {X 0.007,Y -337.994,Z 1653.638,A 0.000,B 0.000,C 90.000,E1 294.823} C_DIS
LIN {X 0.145,Y -352.538,Z 1653.628,A 0.000,B 0.000,C 90.000,E1 292.950} C_DIS
LIN {X 0.097,Y -367.011,Z 1653.618,A 0.000,B 0.000,C 90.000,E1 291.153} C_DIS
LIN {X -0.139,Y -374.027,Z 1653.613,A 0.000,B 0.000,C 90.000,E1 290.301} C_DIS
LIN {X 0.052,Y -380.651,Z 1653.608,A 0.000,B 0.000,C 90.000,E1 289.396} C_DIS
LIN {X -0.060,Y -386.711,Z 1653.603,A 0.000,B 0.000,C 90.000,E1 288.544} C_DIS
LIN {X -0.113,Y -392.176,Z 1653.598,A 0.000,B 0.000,C 90.000,E1 287.692} C_DIS
LIN {X 0.135,Y -396.838,Z 1653.594,A 0.000,B 0.000,C 90.000,E1 286.804} C_DIS
LIN {X 0.059,Y -400.618,Z 1653.589,A 0.000,B 0.000,C 90.000,E1 285.969} C_DIS
LIN {X 0.014,Y -403.529,Z 1653.584,A 0.000,B 0.000,C 90.000,E1 285.134} C_DIS
LIN {X -0.103,Y -405.010,Z 1653.581,A 0.000,B 0.000,C 90.000,E1 284.592} C_DIS
LIN {X 0.081,Y -406.100,Z 1653.578,A 0.000,B 0.000,C 90.000,E1 284.008} C_DIS
LIN {X -0.023,Y -406.762,Z 1653.575,A 0.000,B 0.000,C 90.000,E1 283.467} C_DIS
LIN {X 0.180,Y -407.008,Z 1653.572,A 0.000,B 0.000,C 90.000,E1 282.883} C_DIS
LIN {X -0.010,Y -406.712,Z 1653.569,A 0.000,B 0.000,C 90.000,E1 282.355} C_DIS
LIN {X 0.200,Y -405.960,Z 1653.566,A 0.000,B 0.000,C 90.000,E1 281.771} C_DIS
LIN {X 0.010,Y -404.649,Z 1653.563,A 0.000,B 0.000,C 90.000,E1 281.243} C_DIS
LIN {X 0.211,Y -402.797,Z 1653.559,A 0.000,B 0.000,C 90.000,E1 280.658} C_DIS
LIN {X -0.062,Y -400.319,Z 1653.556,A 0.000,B 0.000,C 90.000,E1 280.141} C_DIS
LIN {X 0.112,Y -397.184,Z 1653.553,A 0.000,B 0.000,C 90.000,E1 279.557} C_DIS
LIN {X -0.123,Y -393.492,Z 1653.550,A 0.000,B 0.000,C 90.000,E1 279.029} C_DIS
LIN {X 0.001,Y -387.217,Z 1653.545,A 0.000,B 0.000,C 90.000,E1 278.163} C_DIS
LIN {X 0.077,Y -380.329,Z 1653.541,A 0.000,B 0.000,C 90.000,E1 277.296} C_DIS
LIN {X 0.074,Y -375.125,Z 1653.537,A 0.000,B 0.000,C 90.000,E1 276.720} C_DIS
LIN {X 0.157,Y -369.344,Z 1653.534,A 0.000,B 0.000,C 90.000,E1 276.144} C_DIS
LIN {X 0.169,Y -363.291,Z 1653.531,A 0.000,B 0.000,C 90.000,E1 275.625} C_DIS
LIN {X 0.130,Y -357.012,Z 1653.529,A 0.000,B 0.000,C 90.000,E1 275.163} C_DIS
LIN {X -0.092,Y -347.333,Z 1653.525,A 0.000,B 0.000,C 90.000,E1 274.588} C_DIS
LIN {X 0.129,Y -337.702,Z 1653.522,A 0.000,B 0.000,C 90.000,E1 274.012} C_DIS
LIN {X -0.013,Y -328.309,Z 1653.520,A 0.000,B 0.000,C 90.000,E1 273.555} C_DIS
LIN {X 0.068,Y -318.438,Z 1653.517,A 0.000,B 0.000,C 90.000,E1 273.094} C_DIS
LIN {X 0.105,Y -308.235,Z 1653.515,A 0.000,B 0.000,C 90.000,E1 272.694} C_DIS
LIN {X 0.103,Y -301.154,Z 1653.514,A 0.000,B 0.000,C 90.000,E1 272.465} C_DIS
LIN {X 0.102,Y -290.196,Z 1653.512,A 0.000,B 0.000,C 90.000,E1 272.178} C_DIS
LIN {X -0.115,Y -282.150,Z 1653.511,A 0.000,B 0.000,C 90.000,E1 272.064} C_DIS
LIN {X 0.094,Y -272.121,Z 1653.511,A 0.000,B 0.000,C 90.000,E1 271.892} C_DIS
LIN {X 0.101,Y -239.209,Z 1653.509,A 0.000,B 0.000,C 90.000,E1 271.661} C_DIS
LIN {X -0.010,Y -200.281,Z 1653.508,A 0.000,B 0.000,C 90.000,E1 271.489} C_DIS
LIN {X 0.043,Y -186.947,Z 1653.508,A 0.000,B 0.000,C 90.000,E1 271.432} C_DIS
LIN {X 0.013,Y -181.364,Z 1653.508,A 0.000,B 0.000,C 90.000,E1 271.432} C_DIS
LIN {X -0.078,Y -181.557,Z 1653.503,A 0.000,B 0.000,C 90.000,E1 270.573} C_DIS
LIN {X 0.032,Y -181.289,Z 1653.494,A 0.000,B 0.000,C 90.000,E1 268.854} C_DIS
LIN {X 0.081,Y -180.907,Z 1653.475,A 0.000,B 0.000,C 90.000,E1 265.469} C_DIS
LIN {X -0.042,Y -180.748,Z 1653.470,A 0.000,B 0.000,C 90.000,E1 264.666} C_DIS
LIN {X 0.026,Y -178.839,Z 1653.442,A 0.000,B 0.000,C 90.000,E1 259.577} C_DIS
LIN {X -0.078,Y -175.883,Z 1653.414,A 0.000,B 0.000,C 90.000,E1 254.519} C_DIS
LIN {X 0.029,Y -174.548,Z 1653.404,A 0.000,B 0.000,C 90.000,E1 252.779} C_DIS
LIN {X -0.038,Y -171.532,Z 1653.381,A 0.000,B 0.000,C 90.000,E1 248.518} C_DIS
LIN {X -0.045,Y -167.758,Z 1653.357,A 0.000,B 0.000,C 90.000,E1 244.204} C_DIS
LIN {X -0.102,Y -166.462,Z 1653.347,A 0.000,B 0.000,C 90.000,E1 242.487} C_DIS
LIN {X 0.035,Y -163.178,Z 1653.328,A 0.000,B 0.000,C 90.000,E1 238.948} C_DIS
LIN {X -0.051,Y -161.138,Z 1653.313,A 0.000,B 0.000,C 90.000,E1 236.342} C_DIS
LIN {X -0.014,Y -157.158,Z 1653.288,A 0.000,B 0.000,C 90.000,E1 231.904} C_DIS
LIN {X 0.009,Y -155.890,Z 1653.278,A 0.000,B 0.000,C 90.000,E1 230.114} C_DIS
LIN {X -0.034,Y -152.140,Z 1653.254,A 0.000,B 0.000,C 90.000,E1 225.648} C_DIS
LIN {X -0.013,Y -150.390,Z 1653.239,A 0.000,B 0.000,C 90.000,E1 222.933} C_DIS
LIN {X 0.011,Y -147.121,Z 1653.213,A 0.000,B 0.000,C 90.000,E1 218.382} C_DIS
LIN {X 0.002,Y -145.685,Z 1653.198,A 0.000,B 0.000,C 90.000,E1 215.644} C_DIS
LIN {X 0.000,Y -143.068,Z 1653.172,A 0.000,B 0.000,C 90.000,E1 211.052} C_DIS
LIN {X -0.069,Y -141.689,Z 1653.152,A 0.000,B 0.000,C 90.000,E1 207.385} C_DIS
LIN {X -0.014,Y -139.460,Z 1653.116,A 0.000,B 0.000,C 90.000,E1 200.865} C_DIS
LIN {X 0.086,Y -139.194,Z 1653.106,A 0.000,B 0.000,C 90.000,E1 198.960} C_DIS
LIN {X -0.027,Y -138.325,Z 1653.054,A 0.000,B 0.000,C 90.000,E1 189.670} C_DIS
LIN {X -0.023,Y -139.452,Z 1653.007,A 0.000,B 0.000,C 90.000,E1 181.260} C_DIS
LIN {X 0.058,Y -140.997,Z 1652.976,A 0.000,B 0.000,C 90.000,E1 175.641} C_DIS
LIN {X 0.007,Y -142.751,Z 1652.955,A 0.000,B 0.000,C 90.000,E1 171.951} C_DIS
LIN {X -0.036,Y -145.152,Z 1652.930,A 0.000,B 0.000,C 90.000,E1 167.353} C_DIS
LIN {X -0.044,Y -147.775,Z 1652.909,A 0.000,B 0.000,C 90.000,E1 163.685} C_DIS
LIN {X 0.036,Y -150.451,Z 1652.889,A 0.000,B 0.000,C 90.000,E1 160.007} C_DIS
LIN {X -0.031,Y -153.899,Z 1652.869,A 0.000,B 0.000,C 90.000,E1 156.410} C_DIS
LIN {X 0.035,Y -157.309,Z 1652.849,A 0.000,B 0.000,C 90.000,E1 152.794} C_DIS
LIN {X -0.018,Y -161.496,Z 1652.829,A 0.000,B 0.000,C 90.000,E1 149.253} C_DIS
LIN {X -0.002,Y -165.696,Z 1652.810,A 0.000,B 0.000,C 90.000,E1 145.722} C_DIS
LIN {X -0.012,Y -170.639,Z 1652.790,A 0.000,B 0.000,C 90.000,E1 142.236} C_DIS
LIN {X 0.038,Y -175.514,Z 1652.771,A 0.000,B 0.000,C 90.000,E1 138.771} C_DIS
END
